LIN {X 0,Y 591.897,Z 1174.931,A -85,B 0,C 180,E1 27089.711,E2 27089.711} C_VEL
LIN {X 0,Y 591.908,Z 1174.109,A -85,B 0,C 180,E1 27087.29,E2 27087.29} C_VEL
LIN {X 0,Y 591.924,Z 1171.503,A -85,B 0,C 180,E1 27084.573,E2 27084.573} C_VEL
LIN {X 0,Y 591.983,Z 1167.392,A -85,B 0,C 180,E1 27082.04,E2 27082.04} C_VEL
LIN {X 0,Y 592.101,Z 1162.202,A -85,B 0,C 180,E1 27079.69,E2 27079.69} C_VEL
LIN {X 0,Y 592.311,Z 1155.916,A -85,B 0,C 180,E1 27077.424,E2 27077.424} C_VEL
LIN {X 0,Y 592.664,Z 1148.61,A -85,B 0,C 180,E1 27075.242,E2 27075.242} C_VEL
LIN {X 0,Y 593.231,Z 1139.207,A -85,B 0,C 180,E1 27072.846,E2 27072.846} C_VEL
LIN {X 0,Y 594.193,Z 1126.707,A -85,B 0,C 180,E1 27070.165,E2 27070.165} C_VEL
LIN {X 0,Y 595.161,Z 1115.669,A -85,B 0,C 180,E1 27068.103,E2 27068.103} C_VEL
LIN {X 0,Y 596.322,Z 1104.081,A -85,B 0,C 180,E1 27066.167,E2 27066.167} C_VEL
LIN {X 0,Y 597.667,Z 1091.843,A -85,B 0,C 180,E1 27064.324,E2 27064.324} C_VEL
LIN {X 0,Y 599.411,Z 1077.454,A -85,B 0,C 180,E1 27062.373,E2 27062.373} C_VEL
LIN {X 0,Y 601.826,Z 1058.389,A -85,B 0,C 180,E1 27060.068,E2 27060.068} C_VEL
LIN {X 0,Y 604.426,Z 1038.878,A -85,B 0,C 180,E1 27058.01,E2 27058.01} C_VEL
LIN {X 0,Y 606.926,Z 1020.464,A -85,B 0,C 180,E1 27056.278,E2 27056.278} C_VEL
LIN {X 0,Y 609.509,Z 1001.423,A -85,B 0,C 180,E1 27054.673,E2 27054.673} C_VEL
LIN {X 0,Y 612.678,Z 977.882,A -85,B 0,C 180,E1 27052.921,E2 27052.921} C_VEL
LIN {X 0,Y 615.57,Z 955.308,A -85,B 0,C 180,E1 27051.472,E2 27051.472} C_VEL
LIN {X 0,Y 618.014,Z 935.338,A -85,B 0,C 180,E1 27050.34,E2 27050.34} C_VEL
LIN {X 0,Y 620.241,Z 915.853,A -85,B 0,C 180,E1 27049.364,E2 27049.364} C_VEL
LIN {X 0,Y 622.411,Z 895.48,A -85,B 0,C 180,E1 27048.471,E2 27048.471} C_VEL
LIN {X 0,Y 624.359,Z 875.247,A -85,B 0,C 180,E1 27047.705,E2 27047.705} C_VEL
LIN {X 0,Y 626.22,Z 853.565,A -85,B 0,C 180,E1 27047.01,E2 27047.01} C_VEL
LIN {X 0,Y 627.748,Z 832.2,A -85,B 0,C 180,E1 27046.449,E2 27046.449} C_VEL
LIN {X 0,Y 629.027,Z 806.934,A -85,B 0,C 180,E1 27045.948,E2 27045.948} C_VEL
LIN {X 0,Y 629.985,Z 765.209,A -85,B 0,C 180,E1 27045.381,E2 27045.381} C_VEL
LIN {X 0,Y 632.547,Z 636.89,A -85,B 0,C 180,E1 27043.662,E2 27043.662} C_VEL
LIN {X 0,Y 637.374,Z 475.557,A -85,B 0,C 180,E1 27041.338,E2 27041.338} C_VEL
LIN {X 0,Y 639.96,Z 392.388,A -85,B 0,C 180,E1 27040.129,E2 27040.129} C_VEL
LIN {X 0,Y 636.531,Z 387.853,A -85,B 0,C 180,E1 27039.678,E2 27039.678} C_VEL
LIN {X 0,Y 622.331,Z 374.151,A -85,B 0,C 180,E1 27037.803,E2 27037.803} C_VEL
LIN {X 0,Y 613.97,Z 366.431,A -85,B 0,C 180,E1 27036.624,E2 27036.624} C_VEL
LIN {X 0,Y 611.495,Z 361.898,A -85,B 0,C 180,E1 27035.323,E2 27035.323} C_VEL
LIN {X 0,Y 608.852,Z 357.084,A -85,B 0,C 180,E1 27033.83,E2 27033.83} C_VEL
LIN {X 0,Y 606.547,Z 352.971,A -85,B 0,C 180,E1 27032.435,E2 27032.435} C_VEL
LIN {X 0,Y 605.226,Z 351.161,A -85,B 0,C 180,E1 27031.693,E2 27031.693} C_VEL
LIN {X 0,Y 602.949,Z 346.733,A -85,B 0,C 180,E1 27030.047,E2 27030.047} C_VEL
LIN {X 0,Y 600.511,Z 343.051,A -85,B 0,C 180,E1 27028.33,E2 27028.33} C_VEL
LIN {X 0,Y 599.929,Z 341.473,A -85,B 0,C 180,E1 27027.711,E2 27027.711} C_VEL
LIN {X 0,Y 597.262,Z 337.966,A -85,B 0,C 180,E1 27025.59,E2 27025.59} C_VEL
LIN {X 0,Y 596.525,Z 335.866,A -85,B 0,C 180,E1 27024.563,E2 27024.563} C_VEL
LIN {X 0,Y 593.473,Z 331.614,A -85,B 0,C 180,E1 27020.927,E2 27020.927} C_VEL
LIN {X 0,Y 593.167,Z 330.296,A -85,B 0,C 180,E1 27019.805,E2 27019.805} C_VEL
LIN {X 0,Y 593.177,Z 330.306,A -85,B 0,C 180,E1 27016.652,E2 27016.652} C_VEL
LIN {X 0,Y 593.194,Z 330.338,A -85,B 0,C 180,E1 27013.451,E2 27013.451} C_VEL
LIN {X 0,Y 593.184,Z 330.295,A -85,B 0,C 180,E1 27010.097,E2 27010.097} C_VEL
LIN {X 0,Y 593.196,Z 330.521,A -85,B 0,C 180,E1 27008.14,E2 27008.14} C_VEL
LIN {X 0,Y 596.195,Z 335.653,A -85,B 0,C 180,E1 27003.943,E2 27003.943} C_VEL
LIN {X 0,Y 596.833,Z 336.421,A -85,B 0,C 180,E1 27003.362,E2 27003.362} C_VEL
LIN {X 0,Y 598.756,Z 340.365,A -85,B 0,C 180,E1 27001.34,E2 27001.34} C_VEL
LIN {X 0,Y 600.215,Z 341.797,A -85,B 0,C 180,E1 27000.382,E2 27000.382} C_VEL
LIN {X 0,Y 601.93,Z 345.619,A -85,B 0,C 180,E1 26998.858,E2 26998.858} C_VEL
LIN {X 0,Y 603.535,Z 347.505,A -85,B 0,C 180,E1 26997.911,E2 26997.911} C_VEL
LIN {X 0,Y 605.549,Z 351.442,A -85,B 0,C 180,E1 26996.497,E2 26996.497} C_VEL
LIN {X 0,Y 606.629,Z 352.745,A -85,B 0,C 180,E1 26995.936,E2 26995.936} C_VEL
LIN {X 0,Y 608.729,Z 356.813,A -85,B 0,C 180,E1 26994.628,E2 26994.628} C_VEL
LIN {X 0,Y 609.804,Z 358.433,A -85,B 0,C 180,E1 26994.071,E2 26994.071} C_VEL
LIN {X 0,Y 612.046,Z 362.396,A -85,B 0,C 180,E1 26992.868,E2 26992.868} C_VEL
LIN {X 0,Y 615.694,Z 369.01,A -85,B 0,C 180,E1 26991.031,E2 26991.031} C_VEL
LIN {X 0,Y 618.78,Z 374.761,A -85,B 0,C 180,E1 26989.573,E2 26989.573} C_VEL
LIN {X 0,Y 621.416,Z 379.7,A -85,B 0,C 180,E1 26988.397,E2 26988.397} C_VEL
LIN {X 0,Y 625.72,Z 387.719,A -85,B 0,C 180,E1 26986.602,E2 26986.602} C_VEL
LIN {X 0,Y 632.277,Z 400.596,A -85,B 0,C 180,E1 26984.028,E2 26984.028} C_VEL
LIN {X 0,Y 638.414,Z 413.491,A -85,B 0,C 180,E1 26981.745,E2 26981.745} C_VEL
LIN {X 0,Y 634.586,Z 446.496,A -85,B 0,C 180,E1 26978.994,E2 26978.994} C_VEL
LIN {X 0,Y 630.632,Z 482.853,A -85,B 0,C 180,E1 26976.102,E2 26976.102} C_VEL
LIN {X 0,Y 626.774,Z 520.74,A -85,B 0,C 180,E1 26973.213,E2 26973.213} C_VEL
LIN {X 0,Y 622.971,Z 560.912,A -85,B 0,C 180,E1 26970.26,E2 26970.26} C_VEL
LIN {X 0,Y 622.003,Z 580.567,A -85,B 0,C 180,E1 26968.779,E2 26968.779} C_VEL
LIN {X 0,Y 622.974,Z 596.183,A -85,B 0,C 180,E1 26967.474,E2 26967.474} C_VEL
LIN {X 0,Y 625.659,Z 609.898,A -85,B 0,C 180,E1 26966.202,E2 26966.202} C_VEL
LIN {X 0,Y 630.378,Z 623.068,A -85,B 0,C 180,E1 26964.845,E2 26964.845} C_VEL
LIN {X 0,Y 637.026,Z 634.807,A -85,B 0,C 180,E1 26963.495,E2 26963.495} C_VEL
LIN {X 0,Y 644.492,Z 643.967,A -85,B 0,C 180,E1 26962.319,E2 26962.319} C_VEL
LIN {X 0,Y 654.158,Z 652.543,A -85,B 0,C 180,E1 26961.081,E2 26961.081} C_VEL
LIN {X 0,Y 665.614,Z 659.76,A -85,B 0,C 180,E1 26959.875,E2 26959.875} C_VEL
LIN {X 0,Y 678.93,Z 665.442,A -85,B 0,C 180,E1 26958.716,E2 26958.716} C_VEL
LIN {X 0,Y 684.652,Z 667.08,A -85,B 0,C 180,E1 26958.244,E2 26958.244} C_VEL
LIN {X 0,Y 688.639,Z 667.261,A -85,B 0,C 180,E1 26957.757,E2 26957.757} C_VEL
LIN {X 0,Y 691.101,Z 666.327,A -85,B 0,C 180,E1 26957.269,E2 26957.269} C_VEL
LIN {X 0,Y 692.176,Z 664.764,A -85,B 0,C 180,E1 26956.842,E2 26956.842} C_VEL
LIN {X 0,Y 684.254,Z 680.558,A -85,B 0,C 180,E1 26956.877,E2 26956.877} C_VEL
LIN {X 0,Y 674.402,Z 696.32,A -85,B 0,C 180,E1 26956.838,E2 26956.838} C_VEL
LIN {X 0,Y 664.605,Z 710.324,A -85,B 0,C 180,E1 26956.682,E2 26956.682} C_VEL
LIN {X 0,Y 657.671,Z 721.169,A -85,B 0,C 180,E1 26956.42,E2 26956.42} C_VEL
LIN {X 0,Y 655.289,Z 724.887,A -85,B 0,C 180,E1 26956.322,E2 26956.322} C_VEL
LIN {X 0,Y 646.984,Z 736.157,A -85,B 0,C 180,E1 26956.067,E2 26956.067} C_VEL
LIN {X 0,Y 640.901,Z 746.673,A -85,B 0,C 180,E1 26955.731,E2 26955.731} C_VEL
LIN {X 0,Y 633.774,Z 760.569,A -85,B 0,C 180,E1 26955.229,E2 26955.229} C_VEL
LIN {X 0,Y 631.455,Z 766.233,A -85,B 0,C 180,E1 26955.02,E2 26955.02} C_VEL
LIN {X 0,Y 629.635,Z 829.003,A -85,B 0,C 180,E1 26954.165,E2 26954.165} C_VEL
LIN {X 0,Y 628.095,Z 857.233,A -85,B 0,C 180,E1 26953.624,E2 26953.624} C_VEL
LIN {X 0,Y 626.337,Z 882.698,A -85,B 0,C 180,E1 26952.976,E2 26952.976} C_VEL
LIN {X 0,Y 624.168,Z 907.973,A -85,B 0,C 180,E1 26952.159,E2 26952.159} C_VEL
LIN {X 0,Y 621.785,Z 932.13,A -85,B 0,C 180,E1 26951.208,E2 26951.208} C_VEL
LIN {X 0,Y 619.008,Z 957.322,A -85,B 0,C 180,E1 26950.034,E2 26950.034} C_VEL
LIN {X 0,Y 616.244,Z 980.499,A -85,B 0,C 180,E1 26948.776,E2 26948.776} C_VEL
LIN {X 0,Y 613.147,Z 1004.437,A -85,B 0,C 180,E1 26947.268,E2 26947.268} C_VEL
LIN {X 0,Y 610.013,Z 1027.671,A -85,B 0,C 180,E1 26945.582,E2 26945.582} C_VEL
LIN {X 0,Y 607.148,Z 1048.872,A -85,B 0,C 180,E1 26943.822,E2 26943.822} C_VEL
LIN {X 0,Y 604.324,Z 1069.852,A -85,B 0,C 180,E1 26941.855,E2 26941.855} C_VEL
LIN {X 0,Y 601.773,Z 1088.672,A -85,B 0,C 180,E1 26939.848,E2 26939.848} C_VEL
LIN {X 0,Y 599.465,Z 1107.176,A -85,B 0,C 180,E1 26937.624,E2 26937.624} C_VEL
LIN {X 0,Y 597.623,Z 1122.284,A -85,B 0,C 180,E1 26935.571,E2 26935.571} C_VEL
LIN {X 0,Y 595.98,Z 1137.726,A -85,B 0,C 180,E1 26933.218,E2 26933.218} C_VEL
LIN {X 0,Y 594.582,Z 1152.188,A -85,B 0,C 180,E1 26930.679,E2 26930.679} C_VEL
LIN {X 0,Y 593.639,Z 1163.642,A -85,B 0,C 180,E1 26928.358,E2 26928.358} C_VEL
LIN {X 0,Y 592.868,Z 1174.752,A -85,B 0,C 180,E1 26925.754,E2 26925.754} C_VEL
LIN {X 0,Y 592.395,Z 1184.279,A -85,B 0,C 180,E1 26923.071,E2 26923.071} C_VEL
LIN {X 0,Y 592.116,Z 1191.662,A -85,B 0,C 180,E1 26920.507,E2 26920.507} C_VEL
LIN {X 0,Y 591.985,Z 1197.33,A -85,B 0,C 180,E1 26917.96,E2 26917.96} C_VEL
LIN {X 0,Y 591.928,Z 1201.413,A -85,B 0,C 180,E1 26915.427,E2 26915.427} C_VEL
LIN {X 0,Y 591.915,Z 1203.98,A -85,B 0,C 180,E1 26912.904,E2 26912.904} C_VEL
LIN {X 0,Y 591.893,Z 1204.916,A -85,B 0,C 180,E1 26910.483,E2 26910.483} C_VEL
LIN {X 0,Y 591.912,Z 1204.414,A -85,B 0,C 180,E1 26907.869,E2 26907.869} C_VEL
LIN {X 0,Y 591.917,Z 1202.356,A -85,B 0,C 180,E1 26905.314,E2 26905.314} C_VEL
LIN {X 0,Y 591.963,Z 1198.771,A -85,B 0,C 180,E1 26902.819,E2 26902.819} C_VEL
LIN {X 0,Y 592.063,Z 1193.554,A -85,B 0,C 180,E1 26900.276,E2 26900.276} C_VEL
LIN {X 0,Y 592.274,Z 1186.734,A -85,B 0,C 180,E1 26897.717,E2 26897.717} C_VEL
LIN {X 0,Y 592.658,Z 1178.841,A -85,B 0,C 180,E1 26895.34,E2 26895.34} C_VEL
LIN {X 0,Y 593.241,Z 1169.012,A -85,B 0,C 180,E1 26892.844,E2 26892.844} C_VEL
LIN {X 0,Y 594.212,Z 1156.49,A -85,B 0,C 180,E1 26890.16,E2 26890.16} C_VEL
LIN {X 0,Y 595.372,Z 1143.738,A -85,B 0,C 180,E1 26887.797,E2 26887.797} C_VEL
LIN {X 0,Y 596.954,Z 1128.582,A -85,B 0,C 180,E1 26885.349,E2 26885.349} C_VEL
LIN {X 0,Y 598.753,Z 1112.617,A -85,B 0,C 180,E1 26883.091,E2 26883.091} C_VEL
LIN {X 0,Y 600.746,Z 1096.868,A -85,B 0,C 180,E1 26881.103,E2 26881.103} C_VEL
LIN {X 0,Y 603.341,Z 1076.831,A -85,B 0,C 180,E1 26878.864,E2 26878.864} C_VEL
LIN {X 0,Y 605.969,Z 1057.522,A -85,B 0,C 180,E1 26876.955,E2 26876.955} C_VEL
LIN {X 0,Y 608.904,Z 1036.067,A -85,B 0,C 180,E1 26875.09,E2 26875.09} C_VEL
LIN {X 0,Y 611.964,Z 1013.202,A -85,B 0,C 180,E1 26873.346,E2 26873.346} C_VEL
LIN {X 0,Y 614.913,Z 990.648,A -85,B 0,C 180,E1 26871.836,E2 26871.836} C_VEL
LIN {X 0,Y 618.022,Z 965.736,A -85,B 0,C 180,E1 26870.398,E2 26870.398} C_VEL
LIN {X 0,Y 620.79,Z 941.484,A -85,B 0,C 180,E1 26869.202,E2 26869.202} C_VEL
LIN {X 0,Y 623.308,Z 916.78,A -85,B 0,C 180,E1 26868.169,E2 26868.169} C_VEL
LIN {X 0,Y 625.72,Z 889.943,A -85,B 0,C 180,E1 26867.242,E2 26867.242} C_VEL
LIN {X 0,Y 627.646,Z 864.672,A -85,B 0,C 180,E1 26866.545,E2 26866.545} C_VEL
LIN {X 0,Y 629.244,Z 837.387,A -85,B 0,C 180,E1 26865.976,E2 26865.976} C_VEL
LIN {X 0,Y 630.409,Z 805.39,A -85,B 0,C 180,E1 26865.494,E2 26865.494} C_VEL
LIN {X 0,Y 631.728,Z 755.195,A -85,B 0,C 180,E1 26864.798,E2 26864.798} C_VEL
LIN {X 0,Y 639.334,Z 659.968,A -85,B 0,C 180,E1 26863.211,E2 26863.211} C_VEL
LIN {X 0,Y 640.721,Z 644.342,A -85,B 0,C 180,E1 26862.962,E2 26862.962} C_VEL
LIN {X 0,Y 643.607,Z 611.399,A -85,B 0,C 180,E1 26862.434,E2 26862.434} C_VEL
LIN {X 0,Y 645.463,Z 593.682,A -85,B 0,C 180,E1 26862.178,E2 26862.178} C_VEL
LIN {X 0,Y 647.573,Z 567.044,A -85,B 0,C 180,E1 26861.731,E2 26861.731} C_VEL
LIN {X 0,Y 651.175,Z 535.673,A -85,B 0,C 180,E1 26861.308,E2 26861.308} C_VEL
LIN {X 0,Y 652.805,Z 513.097,A -85,B 0,C 180,E1 26860.913,E2 26860.913} C_VEL
LIN {X 0,Y 656.784,Z 480.454,A -85,B 0,C 180,E1 26860.496,E2 26860.496} C_VEL
LIN {X 0,Y 657.711,Z 472.636,A -85,B 0,C 180,E1 26860.394,E2 26860.394} C_VEL
LIN {X 0,Y 658.916,Z 453.469,A -85,B 0,C 180,E1 26860.042,E2 26860.042} C_VEL
LIN {X 0,Y 662.468,Z 423.806,A -85,B 0,C 180,E1 26859.659,E2 26859.659} C_VEL
LIN {X 0,Y 662.806,Z 420.787,A -85,B 0,C 180,E1 26859.618,E2 26859.618} C_VEL
LIN {X 0,Y 654.528,Z 413.473,A -85,B 0,C 180,E1 26858.612,E2 26858.612} C_VEL
LIN {X 0,Y 646.489,Z 404.608,A -85,B 0,C 180,E1 26857.545,E2 26857.545} C_VEL
LIN {X 0,Y 630.725,Z 381.497,A -85,B 0,C 180,E1 26855.132,E2 26855.132} C_VEL
LIN {X 0,Y 618.485,Z 364.345,A -85,B 0,C 180,E1 26853.095,E2 26853.095} C_VEL
LIN {X 0,Y 609.724,Z 352.82,A -85,B 0,C 180,E1 26851.543,E2 26851.543} C_VEL
LIN {X 0,Y 605.772,Z 347.565,A -85,B 0,C 180,E1 26850.804,E2 26850.804} C_VEL
LIN {X 0,Y 602.767,Z 343.666,A -85,B 0,C 180,E1 26850.229,E2 26850.229} C_VEL
LIN {X 0,Y 601.685,Z 342.131,A -85,B 0,C 180,E1 26850.014,E2 26850.014} C_VEL
LIN {X 0,Y 598.782,Z 338.928,A -85,B 0,C 180,E1 26849.458,E2 26849.458} C_VEL
LIN {X 0,Y 597.371,Z 336.419,A -85,B 0,C 180,E1 26849.149,E2 26849.149} C_VEL
LIN {X 0,Y 594.578,Z 333.934,A -85,B 0,C 180,E1 26848.614,E2 26848.614} C_VEL
LIN {X 0,Y 593.298,Z 330.916,A -85,B 0,C 180,E1 26848.296,E2 26848.296} C_VEL
LIN {X 0,Y 593.203,Z 330.343,A -85,B 0,C 180,E1 26848.241,E2 26848.241} C_VEL
LIN {X 0,Y 593.175,Z 330.268,A -85,B 0,C 180,E1 26844.921,E2 26844.921} C_VEL
LIN {X 0,Y 593.175,Z 330.342,A -85,B 0,C 180,E1 26841.751,E2 26841.751} C_VEL
LIN {X 0,Y 593.178,Z 330.344,A -85,B 0,C 180,E1 26838.578,E2 26838.578} C_VEL
LIN {X 0,Y 593.172,Z 330.346,A -85,B 0,C 180,E1 26835.376,E2 26835.376} C_VEL
LIN {X 0,Y 593.222,Z 330.489,A -85,B 0,C 180,E1 26834.159,E2 26834.159} C_VEL
LIN {X 0,Y 597.978,Z 346.498,A -85,B 0,C 180,E1 26833.44,E2 26833.44} C_VEL
LIN {X 0,Y 597.928,Z 424.43,A -85,B 0,C 180,E1 26830.722,E2 26830.722} C_VEL
LIN {X 0,Y 598.267,Z 504.666,A -85,B 0,C 180,E1 26827.78,E2 26827.78} C_VEL
LIN {X 0,Y 598.24,Z 578.346,A -85,B 0,C 180,E1 26824.986,E2 26824.986} C_VEL
LIN {X 0,Y 597.772,Z 656.038,A -85,B 0,C 180,E1 26821.965,E2 26821.965} C_VEL
LIN {X 0,Y 597.006,Z 735.74,A -85,B 0,C 180,E1 26818.8,E2 26818.8} C_VEL
LIN {X 0,Y 596.103,Z 814.288,A -85,B 0,C 180,E1 26815.623,E2 26815.623} C_VEL
LIN {X 0,Y 595.528,Z 847.719,A -85,B 0,C 180,E1 26814.267,E2 26814.267} C_VEL
LIN {X 0,Y 595.129,Z 853.977,A -85,B 0,C 180,E1 26814.046,E2 26814.046} C_VEL
LIN {X 0,Y 594.541,Z 967.975,A -85,B 0,C 180,E1 26812.596,E2 26812.596} C_VEL
LIN {X 0,Y 594.552,Z 980.318,A -85,B 0,C 180,E1 26812.313,E2 26812.313} C_VEL
LIN {X 0,Y 594.512,Z 991.961,A -85,B 0,C 180,E1 26811.927,E2 26811.927} C_VEL
LIN {X 0,Y 594.401,Z 1005.064,A -85,B 0,C 180,E1 26811.341,E2 26811.341} C_VEL
LIN {X 0,Y 594.177,Z 1017.894,A -85,B 0,C 180,E1 26810.556,E2 26810.556} C_VEL
LIN {X 0,Y 593.986,Z 1027.459,A -85,B 0,C 180,E1 26809.819,E2 26809.819} C_VEL
LIN {X 0,Y 593.777,Z 1035.869,A -85,B 0,C 180,E1 26809.03,E2 26809.03} C_VEL
LIN {X 0,Y 593.569,Z 1043.67,A -85,B 0,C 180,E1 26808.14,E2 26808.14} C_VEL
LIN {X 0,Y 593.36,Z 1051.4,A -85,B 0,C 180,E1 26807.049,E2 26807.049} C_VEL
LIN {X 0,Y 593.145,Z 1058.271,A -85,B 0,C 180,E1 26805.752,E2 26805.752} C_VEL
LIN {X 0,Y 593.025,Z 1062.584,A -85,B 0,C 180,E1 26804.65,E2 26804.65} C_VEL
LIN {X 0,Y 592.933,Z 1065.672,A -85,B 0,C 180,E1 26803.542,E2 26803.542} C_VEL
LIN {X 0,Y 592.879,Z 1067.603,A -85,B 0,C 180,E1 26802.429,E2 26802.429} C_VEL
LIN {X 0,Y 592.841,Z 1068.45,A -85,B 0,C 180,E1 26801.207,E2 26801.207} C_VEL
LIN {X 0,Y 592.845,Z 1067.619,A -85,B 0,C 180,E1 26799.669,E2 26799.669} C_VEL
LIN {X 0,Y 592.869,Z 1065.357,A -85,B 0,C 180,E1 26798.428,E2 26798.428} C_VEL
LIN {X 0,Y 592.936,Z 1062.021,A -85,B 0,C 180,E1 26797.283,E2 26797.283} C_VEL
LIN {X 0,Y 593.038,Z 1057.325,A -85,B 0,C 180,E1 26796.131,E2 26796.131} C_VEL
LIN {X 0,Y 593.245,Z 1049.74,A -85,B 0,C 180,E1 26794.759,E2 26794.759} C_VEL
LIN {X 0,Y 593.451,Z 1041.883,A -85,B 0,C 180,E1 26793.684,E2 26793.684} C_VEL
LIN {X 0,Y 593.673,Z 1033.295,A -85,B 0,C 180,E1 26792.734,E2 26792.734} C_VEL
LIN {X 0,Y 593.952,Z 1022.469,A -85,B 0,C 180,E1 26791.767,E2 26791.767} C_VEL
LIN {X 0,Y 594.193,Z 1009.805,A -85,B 0,C 180,E1 26790.901,E2 26790.901} C_VEL
LIN {X 0,Y 594.373,Z 998.89,A -85,B 0,C 180,E1 26790.313,E2 26790.313} C_VEL
LIN {X 0,Y 594.504,Z 987.303,A -85,B 0,C 180,E1 26789.825,E2 26789.825} C_VEL
LIN {X 0,Y 594.602,Z 972.83,A -85,B 0,C 180,E1 26789.383,E2 26789.383} C_VEL
LIN {X 0,Y 594.58,Z 956.069,A -85,B 0,C 180,E1 26789.096,E2 26789.096} C_VEL
LIN {X 0,Y 595.087,Z 870.743,A -85,B 0,C 180,E1 26788.038,E2 26788.038} C_VEL
LIN {X 0,Y 594.247,Z 865.604,A -85,B 0,C 180,E1 26787.949,E2 26787.949} C_VEL
LIN {X 0,Y 587.888,Z 851.327,A -85,B 0,C 180,E1 26787.624,E2 26787.624} C_VEL
LIN {X 0,Y 587.567,Z 848.543,A -85,B 0,C 180,E1 26787.539,E2 26787.539} C_VEL
LIN {X 0,Y 588.582,Z 796.208,A -85,B 0,C 180,E1 26785.342,E2 26785.342} C_VEL
LIN {X 0,Y 589.928,Z 714.708,A -85,B 0,C 180,E1 26781.905,E2 26781.905} C_VEL
LIN {X 0,Y 590.88,Z 660.354,A -85,B 0,C 180,E1 26779.6,E2 26779.6} C_VEL
LIN {X 0,Y 592.005,Z 661.931,A -85,B 0,C 180,E1 26779.438,E2 26779.438} C_VEL
LIN {X 0,Y 593.686,Z 661.837,A -85,B 0,C 180,E1 26779.26,E2 26779.26} C_VEL
LIN {X 0,Y 596.517,Z 659.34,A -85,B 0,C 180,E1 26779.018,E2 26779.018} C_VEL
LIN {X 0,Y 600.352,Z 653.293,A -85,B 0,C 180,E1 26778.759,E2 26778.759} C_VEL
LIN {X 0,Y 604.334,Z 651.507,A -85,B 0,C 180,E1 26778.4,E2 26778.4} C_VEL
LIN {X 0,Y 608.324,Z 647.655,A -85,B 0,C 180,E1 26778.106,E2 26778.106} C_VEL
LIN {X 0,Y 611.151,Z 643.737,A -85,B 0,C 180,E1 26777.935,E2 26777.935} C_VEL
LIN {X 0,Y 615.844,Z 641.07,A -85,B 0,C 180,E1 26777.576,E2 26777.576} C_VEL
LIN {X 0,Y 620.545,Z 636.286,A -85,B 0,C 180,E1 26777.253,E2 26777.253} C_VEL
LIN {X 0,Y 622.028,Z 634.442,A -85,B 0,C 180,E1 26777.159,E2 26777.159} C_VEL
LIN {X 0,Y 626.738,Z 631.619,A -85,B 0,C 180,E1 26776.813,E2 26776.813} C_VEL
LIN {X 0,Y 623.646,Z 757.358,A -85,B 0,C 180,E1 26775.063,E2 26775.063} C_VEL
LIN {X 0,Y 622.408,Z 807.519,A -85,B 0,C 180,E1 26774.37,E2 26774.37} C_VEL
LIN {X 0,Y 621.009,Z 834.635,A -85,B 0,C 180,E1 26773.828,E2 26773.828} C_VEL
LIN {X 0,Y 619.62,Z 856.522,A -85,B 0,C 180,E1 26773.27,E2 26773.27} C_VEL
LIN {X 0,Y 618.179,Z 876.153,A -85,B 0,C 180,E1 26772.667,E2 26772.667} C_VEL
LIN {X 0,Y 616.582,Z 893.157,A -85,B 0,C 180,E1 26772.036,E2 26772.036} C_VEL
LIN {X 0,Y 614.249,Z 914.189,A -85,B 0,C 180,E1 26771.121,E2 26771.121} C_VEL
LIN {X 0,Y 612.021,Z 932.876,A -85,B 0,C 180,E1 26770.191,E2 26770.191} C_VEL
LIN {X 0,Y 609.654,Z 951.359,A -85,B 0,C 180,E1 26769.157,E2 26769.157} C_VEL
LIN {X 0,Y 607.2,Z 969.562,A -85,B 0,C 180,E1 26768.016,E2 26768.016} C_VEL
LIN {X 0,Y 604.707,Z 987.416,A -85,B 0,C 180,E1 26766.768,E2 26766.768} C_VEL
LIN {X 0,Y 602.162,Z 1005.245,A -85,B 0,C 180,E1 26765.382,E2 26765.382} C_VEL
LIN {X 0,Y 599.527,Z 1023.571,A -85,B 0,C 180,E1 26763.795,E2 26763.795} C_VEL
LIN {X 0,Y 596.613,Z 1043.916,A -85,B 0,C 180,E1 26761.82,E2 26761.82} C_VEL
LIN {X 0,Y 593.869,Z 1063.27,A -85,B 0,C 180,E1 26759.671,E2 26759.671} C_VEL
LIN {X 0,Y 591.859,Z 1078.36,A -85,B 0,C 180,E1 26757.794,E2 26757.794} C_VEL
LIN {X 0,Y 590.022,Z 1092.656,A -85,B 0,C 180,E1 26755.82,E2 26755.82} C_VEL
LIN {X 0,Y 588.463,Z 1106.104,A -85,B 0,C 180,E1 26753.748,E2 26753.748} C_VEL
LIN {X 0,Y 586.878,Z 1121.364,A -85,B 0,C 180,E1 26751.07,E2 26751.07} C_VEL
LIN {X 0,Y 585.862,Z 1132.457,A -85,B 0,C 180,E1 26748.819,E2 26748.819} C_VEL
LIN {X 0,Y 585.18,Z 1141.293,A -85,B 0,C 180,E1 26746.785,E2 26746.785} C_VEL
LIN {X 0,Y 584.683,Z 1149.344,A -85,B 0,C 180,E1 26744.662,E2 26744.662} C_VEL
LIN {X 0,Y 584.329,Z 1156.234,A -85,B 0,C 180,E1 26742.553,E2 26742.553} C_VEL
LIN {X 0,Y 584.112,Z 1162.464,A -85,B 0,C 180,E1 26740.256,E2 26740.256} C_VEL
LIN {X 0,Y 583.989,Z 1167.597,A -85,B 0,C 180,E1 26737.874,E2 26737.874} C_VEL
LIN {X 0,Y 583.927,Z 1171.885,A -85,B 0,C 180,E1 26735.11,E2 26735.11} C_VEL
LIN {X 0,Y 583.907,Z 1174.164,A -85,B 0,C 180,E1 26732.553,E2 26732.553} C_VEL
LIN {X 0,Y 583.901,Z 1174.928,A -85,B 0,C 180,E1 26730.197,E2 26730.197} C_VEL
LIN {X 0,Y 583.911,Z 1174.355,A -85,B 0,C 180,E1 26727.744,E2 26727.744} C_VEL
LIN {X 0,Y 583.915,Z 1172.492,A -85,B 0,C 180,E1 26725.385,E2 26725.385} C_VEL
LIN {X 0,Y 583.954,Z 1169.172,A -85,B 0,C 180,E1 26722.92,E2 26722.92} C_VEL
LIN {X 0,Y 584.072,Z 1163.675,A -85,B 0,C 180,E1 26720.144,E2 26720.144} C_VEL
LIN {X 0,Y 584.291,Z 1157.111,A -85,B 0,C 180,E1 26717.65,E2 26717.65} C_VEL
LIN {X 0,Y 584.636,Z 1150.02,A -85,B 0,C 180,E1 26715.44,E2 26715.44} C_VEL
LIN {X 0,Y 585.13,Z 1142.068,A -85,B 0,C 180,E1 26713.318,E2 26713.318} C_VEL
LIN {X 0,Y 585.792,Z 1133.335,A -85,B 0,C 180,E1 26711.284,E2 26711.284} C_VEL
LIN {X 0,Y 586.614,Z 1123.912,A -85,B 0,C 180,E1 26709.341,E2 26709.341} C_VEL
LIN {X 0,Y 587.671,Z 1113.33,A -85,B 0,C 180,E1 26707.387,E2 26707.387} C_VEL
LIN {X 0,Y 589.142,Z 1100.183,A -85,B 0,C 180,E1 26705.217,E2 26705.217} C_VEL
LIN {X 0,Y 591.339,Z 1082.2,A -85,B 0,C 180,E1 26702.62,E2 26702.62} C_VEL
LIN {X 0,Y 593.428,Z 1066.615,A -85,B 0,C 180,E1 26700.64,E2 26700.64} C_VEL
LIN {X 0,Y 595.625,Z 1050.692,A -85,B 0,C 180,E1 26698.819,E2 26698.819} C_VEL
LIN {X 0,Y 598.392,Z 1031.392,A -85,B 0,C 180,E1 26696.841,E2 26696.841} C_VEL
LIN {X 0,Y 601.593,Z 1009.292,A -85,B 0,C 180,E1 26694.86,E2 26694.86} C_VEL
LIN {X 0,Y 604.36,Z 989.93,A -85,B 0,C 180,E1 26693.328,E2 26693.328} C_VEL
LIN {X 0,Y 606.925,Z 971.551,A -85,B 0,C 180,E1 26692.026,E2 26692.026} C_VEL
LIN {X 0,Y 609.36,Z 953.557,A -85,B 0,C 180,E1 26690.884,E2 26690.884} C_VEL
LIN {X 0,Y 611.705,Z 935.317,A -85,B 0,C 180,E1 26689.848,E2 26689.848} C_VEL
LIN {X 0,Y 614.049,Z 915.832,A -85,B 0,C 180,E1 26688.866,E2 26688.866} C_VEL
LIN {X 0,Y 616.241,Z 896.216,A -85,B 0,C 180,E1 26687.999,E2 26687.999} C_VEL
LIN {X 0,Y 617.87,Z 879.929,A -85,B 0,C 180,E1 26687.373,E2 26687.373} C_VEL
LIN {X 0,Y 619.415,Z 859.522,A -85,B 0,C 180,E1 26686.725,E2 26686.725} C_VEL
LIN {X 0,Y 620.797,Z 838.049,A -85,B 0,C 180,E1 26686.164,E2 26686.164} C_VEL
LIN {X 0,Y 621.872,Z 817.652,A -85,B 0,C 180,E1 26685.73,E2 26685.73} C_VEL
LIN {X 0,Y 622.665,Z 798.147,A -85,B 0,C 180,E1 26685.403,E2 26685.403} C_VEL
LIN {X 0,Y 626.399,Z 642.254,A -85,B 0,C 180,E1 26683.253,E2 26683.253} C_VEL
LIN {X 0,Y 634.16,Z 414.07,A -85,B 0,C 180,E1 26679.889,E2 26679.889} C_VEL
LIN {X 0,Y 634.628,Z 396.39,A -85,B 0,C 180,E1 26679.621,E2 26679.621} C_VEL
LIN {X 0,Y 632.055,Z 393.601,A -85,B 0,C 180,E1 26679.286,E2 26679.286} C_VEL
LIN {X 0,Y 619.781,Z 381.516,A -85,B 0,C 180,E1 26677.636,E2 26677.636} C_VEL
LIN {X 0,Y 611.282,Z 373.672,A -85,B 0,C 180,E1 26676.425,E2 26676.425} C_VEL
LIN {X 0,Y 608.132,Z 370.809,A -85,B 0,C 180,E1 26675.943,E2 26675.943} C_VEL
LIN {X 0,Y 606.822,Z 368.308,A -85,B 0,C 180,E1 26675.22,E2 26675.22} C_VEL
LIN {X 0,Y 604.105,Z 363.41,A -85,B 0,C 180,E1 26673.675,E2 26673.675} C_VEL
LIN {X 0,Y 601.839,Z 359.085,A -85,B 0,C 180,E1 26672.229,E2 26672.229} C_VEL
LIN {X 0,Y 599.198,Z 354.948,A -85,B 0,C 180,E1 26670.568,E2 26670.568} C_VEL
LIN {X 0,Y 598.463,Z 353.328,A -85,B 0,C 180,E1 26669.971,E2 26669.971} C_VEL
LIN {X 0,Y 596.055,Z 349.621,A -85,B 0,C 180,E1 26668.233,E2 26668.233} C_VEL
LIN {X 0,Y 595.332,Z 347.979,A -85,B 0,C 180,E1 26667.53,E2 26667.53} C_VEL
LIN {X 0,Y 592.79,Z 344.325,A -85,B 0,C 180,E1 26665.368,E2 26665.368} C_VEL
LIN {X 0,Y 592.163,Z 342.565,A -85,B 0,C 180,E1 26664.483,E2 26664.483} C_VEL
LIN {X 0,Y 589.172,Z 338.216,A -85,B 0,C 180,E1 26660.76,E2 26660.76} C_VEL
LIN {X 0,Y 588.742,Z 336.959,A -85,B 0,C 180,E1 26659.65,E2 26659.65} C_VEL
LIN {X 0,Y 587.04,Z 335.405,A -85,B 0,C 180,E1 26655.005,E2 26655.005} C_VEL
LIN {X 0,Y 587.489,Z 335.904,A -85,B 0,C 180,E1 26651.088,E2 26651.088} C_VEL
LIN {X 0,Y 588.982,Z 337.422,A -85,B 0,C 180,E1 26648.1,E2 26648.1} C_VEL
LIN {X 0,Y 592.051,Z 342.514,A -85,B 0,C 180,E1 26643.874,E2 26643.874} C_VEL
LIN {X 0,Y 592.582,Z 343.466,A -85,B 0,C 180,E1 26643.289,E2 26643.289} C_VEL
LIN {X 0,Y 594.754,Z 347.428,A -85,B 0,C 180,E1 26641.156,E2 26641.156} C_VEL
LIN {X 0,Y 595.851,Z 348.705,A -85,B 0,C 180,E1 26640.385,E2 26640.385} C_VEL
LIN {X 0,Y 597.8,Z 352.589,A -85,B 0,C 180,E1 26638.754,E2 26638.754} C_VEL
LIN {X 0,Y 599.06,Z 354.138,A -85,B 0,C 180,E1 26637.991,E2 26637.991} C_VEL
LIN {X 0,Y 601.26,Z 358.247,A -85,B 0,C 180,E1 26636.472,E2 26636.472} C_VEL
LIN {X 0,Y 602.214,Z 359.757,A -85,B 0,C 180,E1 26635.906,E2 26635.906} C_VEL
LIN {X 0,Y 604.639,Z 363.873,A -85,B 0,C 180,E1 26634.496,E2 26634.496} C_VEL
LIN {X 0,Y 607.579,Z 369.036,A -85,B 0,C 180,E1 26632.894,E2 26632.894} C_VEL
LIN {X 0,Y 611.111,Z 375.716,A -85,B 0,C 180,E1 26631.058,E2 26631.058} C_VEL
LIN {X 0,Y 614.004,Z 381.082,A -85,B 0,C 180,E1 26629.681,E2 26629.681} C_VEL
LIN {X 0,Y 618.347,Z 389.075,A -85,B 0,C 180,E1 26627.77,E2 26627.77} C_VEL
LIN {X 0,Y 625.086,Z 402.367,A -85,B 0,C 180,E1 26624.981,E2 26624.981} C_VEL
LIN {X 0,Y 631.564,Z 415.802,A -85,B 0,C 180,E1 26622.494,E2 26622.494} C_VEL
LIN {X 0,Y 632.751,Z 418.495,A -85,B 0,C 180,E1 26622.038,E2 26622.038} C_VEL
LIN {X 0,Y 628.808,Z 450.791,A -85,B 0,C 180,E1 26619.328,E2 26619.328} C_VEL
LIN {X 0,Y 624.705,Z 486.494,A -85,B 0,C 180,E1 26616.468,E2 26616.468} C_VEL
LIN {X 0,Y 620.615,Z 524.504,A -85,B 0,C 180,E1 26613.546,E2 26613.546} C_VEL
LIN {X 0,Y 616.585,Z 564.906,A -85,B 0,C 180,E1 26610.551,E2 26610.551} C_VEL
LIN {X 0,Y 615.611,Z 583.676,A -85,B 0,C 180,E1 26609.119,E2 26609.119} C_VEL
LIN {X 0,Y 616.536,Z 599.846,A -85,B 0,C 180,E1 26607.753,E2 26607.753} C_VEL
LIN {X 0,Y 619.371,Z 614.497,A -85,B 0,C 180,E1 26606.377,E2 26606.377} C_VEL
LIN {X 0,Y 624.083,Z 627.709,A -85,B 0,C 180,E1 26605,E2 26605} C_VEL
LIN {X 0,Y 630.665,Z 639.502,A -85,B 0,C 180,E1 26603.632,E2 26603.632} C_VEL
LIN {X 0,Y 638.042,Z 648.781,A -85,B 0,C 180,E1 26602.438,E2 26602.438} C_VEL
LIN {X 0,Y 647.588,Z 657.546,A -85,B 0,C 180,E1 26601.18,E2 26601.18} C_VEL
LIN {X 0,Y 658.908,Z 664.997,A -85,B 0,C 180,E1 26599.953,E2 26599.953} C_VEL
LIN {X 0,Y 671.336,Z 670.726,A -85,B 0,C 180,E1 26598.828,E2 26598.828} C_VEL
LIN {X 0,Y 680.797,Z 673.766,A -85,B 0,C 180,E1 26598.067,E2 26598.067} C_VEL
LIN {X 0,Y 684.978,Z 674.105,A -85,B 0,C 180,E1 26597.592,E2 26597.592} C_VEL
LIN {X 0,Y 685.455,Z 674.112,A -85,B 0,C 180,E1 26597.515,E2 26597.515} C_VEL
LIN {X 0,Y 674.505,Z 689.052,A -85,B 0,C 180,E1 26597.453,E2 26597.453} C_VEL
LIN {X 0,Y 661.923,Z 704.601,A -85,B 0,C 180,E1 26597.232,E2 26597.232} C_VEL
LIN {X 0,Y 653.836,Z 716.002,A -85,B 0,C 180,E1 26596.967,E2 26596.967} C_VEL
LIN {X 0,Y 649.863,Z 722.315,A -85,B 0,C 180,E1 26596.789,E2 26596.789} C_VEL
LIN {X 0,Y 641.335,Z 733.878,A -85,B 0,C 180,E1 26596.529,E2 26596.529} C_VEL
LIN {X 0,Y 635.156,Z 744.353,A -85,B 0,C 180,E1 26596.2,E2 26596.2} C_VEL
LIN {X 0,Y 627.217,Z 759.808,A -85,B 0,C 180,E1 26595.639,E2 26595.639} C_VEL
LIN {X 0,Y 626.243,Z 762.541,A -85,B 0,C 180,E1 26595.555,E2 26595.555} C_VEL
LIN {X 0,Y 625.47,Z 772.425,A -85,B 0,C 180,E1 26595.471,E2 26595.471} C_VEL
LIN {X 0,Y 623.944,Z 827.243,A -85,B 0,C 180,E1 26594.703,E2 26594.703} C_VEL
LIN {X 0,Y 622.273,Z 855.617,A -85,B 0,C 180,E1 26594.161,E2 26594.161} C_VEL
LIN {X 0,Y 620.284,Z 882.798,A -85,B 0,C 180,E1 26593.467,E2 26593.467} C_VEL
LIN {X 0,Y 618.078,Z 908.548,A -85,B 0,C 180,E1 26592.641,E2 26592.641} C_VEL
LIN {X 0,Y 615.728,Z 931.388,A -85,B 0,C 180,E1 26591.742,E2 26591.742} C_VEL
LIN {X 0,Y 612.797,Z 956.795,A -85,B 0,C 180,E1 26590.556,E2 26590.556} C_VEL
LIN {X 0,Y 609.827,Z 980.503,A -85,B 0,C 180,E1 26589.262,E2 26589.262} C_VEL
LIN {X 0,Y 606.706,Z 1003.411,A -85,B 0,C 180,E1 26587.81,E2 26587.81} C_VEL
LIN {X 0,Y 603.443,Z 1026.315,A -85,B 0,C 180,E1 26586.147,E2 26586.147} C_VEL
LIN {X 0,Y 600.359,Z 1047.699,A -85,B 0,C 180,E1 26584.372,E2 26584.372} C_VEL
LIN {X 0,Y 597.368,Z 1068.839,A -85,B 0,C 180,E1 26582.384,E2 26582.384} C_VEL
LIN {X 0,Y 594.562,Z 1088.261,A -85,B 0,C 180,E1 26580.297,E2 26580.297} C_VEL
LIN {X 0,Y 592.13,Z 1106.396,A -85,B 0,C 180,E1 26578.106,E2 26578.106} C_VEL
LIN {X 0,Y 590.073,Z 1122.283,A -85,B 0,C 180,E1 26575.923,E2 26575.923} C_VEL
LIN {X 0,Y 588.307,Z 1137.724,A -85,B 0,C 180,E1 26573.539,E2 26573.539} C_VEL
LIN {X 0,Y 586.809,Z 1152.191,A -85,B 0,C 180,E1 26570.965,E2 26570.965} C_VEL
LIN {X 0,Y 585.747,Z 1164.11,A -85,B 0,C 180,E1 26568.511,E2 26568.511} C_VEL
LIN {X 0,Y 584.957,Z 1174.75,A -85,B 0,C 180,E1 26565.973,E2 26565.973} C_VEL
LIN {X 0,Y 584.44,Z 1184.277,A -85,B 0,C 180,E1 26563.252,E2 26563.252} C_VEL
LIN {X 0,Y 584.131,Z 1191.663,A -85,B 0,C 180,E1 26560.652,E2 26560.652} C_VEL
LIN {X 0,Y 583.989,Z 1197.329,A -85,B 0,C 180,E1 26558.07,E2 26558.07} C_VEL
LIN {X 0,Y 583.929,Z 1201.412,A -85,B 0,C 180,E1 26555.501,E2 26555.501} C_VEL
LIN {X 0,Y 583.916,Z 1203.979,A -85,B 0,C 180,E1 26552.943,E2 26552.943} C_VEL
LIN {X 0,Y 583.893,Z 1204.916,A -85,B 0,C 180,E1 26550.489,E2 26550.489} C_VEL
LIN {X 0,Y 583.911,Z 1204.413,A -85,B 0,C 180,E1 26547.84,E2 26547.84} C_VEL
LIN {X 0,Y 583.918,Z 1202.391,A -85,B 0,C 180,E1 26545.282,E2 26545.282} C_VEL
LIN {X 0,Y 583.97,Z 1198.769,A -85,B 0,C 180,E1 26542.72,E2 26542.72} C_VEL
LIN {X 0,Y 584.075,Z 1193.552,A -85,B 0,C 180,E1 26540.142,E2 26540.142} C_VEL
LIN {X 0,Y 584.31,Z 1186.733,A -85,B 0,C 180,E1 26537.547,E2 26537.547} C_VEL
LIN {X 0,Y 584.744,Z 1178.486,A -85,B 0,C 180,E1 26535.035,E2 26535.035} C_VEL
LIN {X 0,Y 585.394,Z 1168.583,A -85,B 0,C 180,E1 26532.504,E2 26532.504} C_VEL
LIN {X 0,Y 586.407,Z 1156.328,A -85,B 0,C 180,E1 26529.852,E2 26529.852} C_VEL
LIN {X 0,Y 587.714,Z 1143.159,A -85,B 0,C 180,E1 26527.386,E2 26527.386} C_VEL
LIN {X 0,Y 589.512,Z 1127.255,A -85,B 0,C 180,E1 26524.802,E2 26524.802} C_VEL
LIN {X 0,Y 591.49,Z 1111.057,A -85,B 0,C 180,E1 26522.516,E2 26522.516} C_VEL
LIN {X 0,Y 593.856,Z 1093.671,A -85,B 0,C 180,E1 26520.32,E2 26520.32} C_VEL
LIN {X 0,Y 596.511,Z 1074.442,A -85,B 0,C 180,E1 26518.196,E2 26518.196} C_VEL
LIN {X 0,Y 599.557,Z 1053.51,A -85,B 0,C 180,E1 26516.149,E2 26516.149} C_VEL
LIN {X 0,Y 602.708,Z 1031.646,A -85,B 0,C 180,E1 26514.269,E2 26514.269} C_VEL
LIN {X 0,Y 605.837,Z 1009.375,A -85,B 0,C 180,E1 26512.601,E2 26512.601} C_VEL
LIN {X 0,Y 608.985,Z 986.501,A -85,B 0,C 180,E1 26511.102,E2 26511.102} C_VEL
LIN {X 0,Y 612.195,Z 961.744,A -85,B 0,C 180,E1 26509.7,E2 26509.7} C_VEL
LIN {X 0,Y 615.047,Z 937.979,A -85,B 0,C 180,E1 26508.543,E2 26508.543} C_VEL
LIN {X 0,Y 617.507,Z 914.255,A -85,B 0,C 180,E1 26507.569,E2 26507.569} C_VEL
LIN {X 0,Y 619.905,Z 887.591,A -85,B 0,C 180,E1 26506.673,E2 26506.673} C_VEL
LIN {X 0,Y 621.996,Z 860.208,A -85,B 0,C 180,E1 26505.942,E2 26505.942} C_VEL
LIN {X 0,Y 623.686,Z 832.533,A -85,B 0,C 180,E1 26505.383,E2 26505.383} C_VEL
LIN {X 0,Y 624.899,Z 797.21,A -85,B 0,C 180,E1 26504.866,E2 26504.866} C_VEL
LIN {X 0,Y 626.19,Z 751.211,A -85,B 0,C 180,E1 26504.227,E2 26504.227} C_VEL
LIN {X 0,Y 633.652,Z 660.134,A -85,B 0,C 180,E1 26502.704,E2 26502.704} C_VEL
LIN {X 0,Y 635.032,Z 644.759,A -85,B 0,C 180,E1 26502.457,E2 26502.457} C_VEL
LIN {X 0,Y 638.008,Z 611.522,A -85,B 0,C 180,E1 26501.923,E2 26501.923} C_VEL
LIN {X 0,Y 639.842,Z 594.136,A -85,B 0,C 180,E1 26501.67,E2 26501.67} C_VEL
LIN {X 0,Y 642.055,Z 567.049,A -85,B 0,C 180,E1 26501.215,E2 26501.215} C_VEL
LIN {X 0,Y 645.629,Z 536.228,A -85,B 0,C 180,E1 26500.798,E2 26500.798} C_VEL
LIN {X 0,Y 647.373,Z 513.052,A -85,B 0,C 180,E1 26500.394,E2 26500.394} C_VEL
LIN {X 0,Y 651.452,Z 480.082,A -85,B 0,C 180,E1 26499.974,E2 26499.974} C_VEL
LIN {X 0,Y 652.249,Z 473.101,A -85,B 0,C 180,E1 26499.879,E2 26499.879} C_VEL
LIN {X 0,Y 653.585,Z 453.267,A -85,B 0,C 180,E1 26499.517,E2 26499.517} C_VEL
LIN {X 0,Y 656.819,Z 425.778,A -85,B 0,C 180,E1 26499.153,E2 26499.153} C_VEL
LIN {X 0,Y 645.344,Z 414.407,A -85,B 0,C 180,E1 26497.679,E2 26497.679} C_VEL
LIN {X 0,Y 638.653,Z 405.195,A -85,B 0,C 180,E1 26496.704,E2 26496.704} C_VEL
LIN {X 0,Y 625.051,Z 385.145,A -85,B 0,C 180,E1 26494.548,E2 26494.548} C_VEL
LIN {X 0,Y 614.266,Z 370.144,A -85,B 0,C 180,E1 26492.713,E2 26492.713} C_VEL
LIN {X 0,Y 606.187,Z 359.352,A -85,B 0,C 180,E1 26491.249,E2 26491.249} C_VEL
LIN {X 0,Y 602.382,Z 354.271,A -85,B 0,C 180,E1 26490.526,E2 26490.526} C_VEL
LIN {X 0,Y 599.108,Z 349.769,A -85,B 0,C 180,E1 26489.88,E2 26489.88} C_VEL
LIN {X 0,Y 595.371,Z 345.396,A -85,B 0,C 180,E1 26489.146,E2 26489.146} C_VEL
LIN {X 0,Y 594.142,Z 343.451,A -85,B 0,C 180,E1 26488.881,E2 26488.881} C_VEL
LIN {X 0,Y 591.204,Z 340.396,A -85,B 0,C 180,E1 26488.293,E2 26488.293} C_VEL
LIN {X 0,Y 589.555,Z 337.457,A -85,B 0,C 180,E1 26487.911,E2 26487.911} C_VEL
LIN {X 0,Y 586.738,Z 335.031,A -85,B 0,C 180,E1 26487.34,E2 26487.34} C_VEL
LIN {X 0,Y 585.356,Z 331.986,A -85,B 0,C 180,E1 26486.984,E2 26486.984} C_VEL
LIN {X 0,Y 585.234,Z 331.272,A -85,B 0,C 180,E1 26486.921,E2 26486.921} C_VEL
LIN {X 0,Y 585.254,Z 331.289,A -85,B 0,C 180,E1 26483.565,E2 26483.565} C_VEL
LIN {X 0,Y 585.253,Z 331.312,A -85,B 0,C 180,E1 26480.289,E2 26480.289} C_VEL
LIN {X 0,Y 585.252,Z 331.31,A -85,B 0,C 180,E1 26476.987,E2 26476.987} C_VEL
LIN {X 0,Y 585.266,Z 331.347,A -85,B 0,C 180,E1 26474.421,E2 26474.421} C_VEL
LIN {X 0,Y 590.441,Z 347.93,A -85,B 0,C 180,E1 26473.665,E2 26473.665} C_VEL
LIN {X 0,Y 590.332,Z 429.486,A -85,B 0,C 180,E1 26470.802,E2 26470.802} C_VEL
LIN {X 0,Y 590.654,Z 510.012,A -85,B 0,C 180,E1 26467.832,E2 26467.832} C_VEL
LIN {X 0,Y 590.573,Z 585.574,A -85,B 0,C 180,E1 26464.954,E2 26464.954} C_VEL
LIN {X 0,Y 590,Z 663.403,A -85,B 0,C 180,E1 26461.894,E2 26461.894} C_VEL
LIN {X 0,Y 589.426,Z 724.729,A -85,B 0,C 180,E1 26459.465,E2 26459.465} C_VEL
LIN {X 0,Y 588.503,Z 802.993,A -85,B 0,C 180,E1 26456.298,E2 26456.298} C_VEL
LIN {X 0,Y 587.72,Z 848.985,A -85,B 0,C 180,E1 26454.424,E2 26454.424} C_VEL
LIN {X 0,Y 587.314,Z 855.326,A -85,B 0,C 180,E1 26454.2,E2 26454.2} C_VEL
LIN {X 0,Y 586.692,Z 969.277,A -85,B 0,C 180,E1 26452.724,E2 26452.724} C_VEL
LIN {X 0,Y 586.71,Z 981.563,A -85,B 0,C 180,E1 26452.438,E2 26452.438} C_VEL
LIN {X 0,Y 586.672,Z 993.42,A -85,B 0,C 180,E1 26452.038,E2 26452.038} C_VEL
LIN {X 0,Y 586.55,Z 1006.901,A -85,B 0,C 180,E1 26451.422,E2 26451.422} C_VEL
LIN {X 0,Y 586.332,Z 1018.871,A -85,B 0,C 180,E1 26450.677,E2 26450.677} C_VEL
LIN {X 0,Y 586.132,Z 1028.481,A -85,B 0,C 180,E1 26449.93,E2 26449.93} C_VEL
LIN {X 0,Y 585.927,Z 1036.447,A -85,B 0,C 180,E1 26449.18,E2 26449.18} C_VEL
LIN {X 0,Y 585.705,Z 1044.353,A -85,B 0,C 180,E1 26448.279,E2 26448.279} C_VEL
LIN {X 0,Y 585.496,Z 1051.508,A -85,B 0,C 180,E1 26447.273,E2 26447.273} C_VEL
LIN {X 0,Y 585.273,Z 1058.751,A -85,B 0,C 180,E1 26445.96,E2 26445.96} C_VEL
LIN {X 0,Y 585.121,Z 1063.55,A -85,B 0,C 180,E1 26444.742,E2 26444.742} C_VEL
LIN {X 0,Y 585.02,Z 1066.686,A -85,B 0,C 180,E1 26443.62,E2 26443.62} C_VEL
LIN {X 0,Y 584.961,Z 1068.658,A -85,B 0,C 180,E1 26442.492,E2 26442.492} C_VEL
LIN {X 0,Y 584.92,Z 1069.508,A -85,B 0,C 180,E1 26441.357,E2 26441.357} C_VEL
LIN {X 0,Y 584.915,Z 1069.157,A -85,B 0,C 180,E1 26440.087,E2 26440.087} C_VEL
LIN {X 0,Y 584.947,Z 1066.794,A -85,B 0,C 180,E1 26438.543,E2 26438.543} C_VEL
LIN {X 0,Y 585.016,Z 1063.509,A -85,B 0,C 180,E1 26437.362,E2 26437.362} C_VEL
LIN {X 0,Y 585.115,Z 1059.021,A -85,B 0,C 180,E1 26436.216,E2 26436.216} C_VEL
LIN {X 0,Y 585.282,Z 1052.953,A -85,B 0,C 180,E1 26435.041,E2 26435.041} C_VEL
LIN {X 0,Y 585.537,Z 1044.166,A -85,B 0,C 180,E1 26433.75,E2 26433.75} C_VEL
LIN {X 0,Y 585.769,Z 1035.678,A -85,B 0,C 180,E1 26432.776,E2 26432.776} C_VEL
LIN {X 0,Y 586.014,Z 1026.375,A -85,B 0,C 180,E1 26431.905,E2 26431.905} C_VEL
LIN {X 0,Y 586.271,Z 1014.814,A -85,B 0,C 180,E1 26431.029,E2 26431.029} C_VEL
LIN {X 0,Y 586.509,Z 1001.364,A -85,B 0,C 180,E1 26430.257,E2 26430.257} C_VEL
LIN {X 0,Y 586.649,Z 990.146,A -85,B 0,C 180,E1 26429.763,E2 26429.763} C_VEL
LIN {X 0,Y 586.732,Z 977.999,A -85,B 0,C 180,E1 26429.363,E2 26429.363} C_VEL
LIN {X 0,Y 586.757,Z 963.626,A -85,B 0,C 180,E1 26429.044,E2 26429.044} C_VEL
LIN {X 0,Y 587.49,Z 849.557,A -85,B 0,C 180,E1 26427.58,E2 26427.58} C_VEL
LIN {X 0,Y 587.567,Z 848.543,A -85,B 0,C 180,E1 26427.539,E2 26427.539} C_VEL
LIN {X 0,Y 587.224,Z 842.494,A -85,B 0,C 180,E1 26427.273,E2 26427.273} C_VEL
LIN {X 0,Y 584.341,Z 832.92,A -85,B 0,C 180,E1 26426.786,E2 26426.786} C_VEL
LIN {X 0,Y 581.014,Z 822.38,A -85,B 0,C 180,E1 26426.242,E2 26426.242} C_VEL
LIN {X 0,Y 580.535,Z 817.332,A -85,B 0,C 180,E1 26426.012,E2 26426.012} C_VEL
LIN {X 0,Y 581.909,Z 735.659,A -85,B 0,C 180,E1 26422.548,E2 26422.548} C_VEL
LIN {X 0,Y 583.027,Z 677.37,A -85,B 0,C 180,E1 26420.053,E2 26420.053} C_VEL
LIN {X 0,Y 584.211,Z 678.898,A -85,B 0,C 180,E1 26419.88,E2 26419.88} C_VEL
LIN {X 0,Y 586.069,Z 678.582,A -85,B 0,C 180,E1 26419.681,E2 26419.681} C_VEL
LIN {X 0,Y 589.016,Z 675.686,A -85,B 0,C 180,E1 26419.43,E2 26419.43} C_VEL
LIN {X 0,Y 592.682,Z 669.871,A -85,B 0,C 180,E1 26419.176,E2 26419.176} C_VEL
LIN {X 0,Y 596.077,Z 668.392,A -85,B 0,C 180,E1 26418.854,E2 26418.854} C_VEL
LIN {X 0,Y 599.972,Z 664.609,A -85,B 0,C 180,E1 26418.544,E2 26418.544} C_VEL
LIN {X 0,Y 603.114,Z 660.169,A -85,B 0,C 180,E1 26418.332,E2 26418.332} C_VEL
LIN {X 0,Y 607.776,Z 657.362,A -85,B 0,C 180,E1 26417.965,E2 26417.965} C_VEL
LIN {X 0,Y 612.66,Z 652.272,A -85,B 0,C 180,E1 26417.636,E2 26417.636} C_VEL
LIN {X 0,Y 614.453,Z 650.24,A -85,B 0,C 180,E1 26417.52,E2 26417.52} C_VEL
LIN {X 0,Y 619.851,Z 646.474,A -85,B 0,C 180,E1 26417.13,E2 26417.13} C_VEL
LIN {X 0,Y 620.331,Z 646.144,A -85,B 0,C 180,E1 26417.095,E2 26417.095} C_VEL
LIN {X 0,Y 616.972,Z 766.217,A -85,B 0,C 180,E1 26415.379,E2 26415.379} C_VEL
LIN {X 0,Y 615.721,Z 809.824,A -85,B 0,C 180,E1 26414.756,E2 26414.756} C_VEL
LIN {X 0,Y 614.29,Z 836.155,A -85,B 0,C 180,E1 26414.213,E2 26414.213} C_VEL
LIN {X 0,Y 612.796,Z 858.535,A -85,B 0,C 180,E1 26413.629,E2 26413.629} C_VEL
LIN {X 0,Y 611.04,Z 881.488,A -85,B 0,C 180,E1 26412.902,E2 26412.902} C_VEL
LIN {X 0,Y 608.576,Z 909.082,A -85,B 0,C 180,E1 26411.841,E2 26411.841} C_VEL
LIN {X 0,Y 606.288,Z 929.004,A -85,B 0,C 180,E1 26410.9,E2 26410.9} C_VEL
LIN {X 0,Y 603.515,Z 949.631,A -85,B 0,C 180,E1 26409.756,E2 26409.756} C_VEL
LIN {X 0,Y 600.787,Z 968.864,A -85,B 0,C 180,E1 26408.551,E2 26408.551} C_VEL
LIN {X 0,Y 598.057,Z 987.419,A -85,B 0,C 180,E1 26407.246,E2 26407.246} C_VEL
LIN {X 0,Y 595.288,Z 1005.767,A -85,B 0,C 180,E1 26405.805,E2 26405.805} C_VEL
LIN {X 0,Y 592.5,Z 1024.151,A -85,B 0,C 180,E1 26404.192,E2 26404.192} C_VEL
LIN {X 0,Y 589.259,Z 1045.522,A -85,B 0,C 180,E1 26402.082,E2 26402.082} C_VEL
LIN {X 0,Y 586.446,Z 1064.144,A -85,B 0,C 180,E1 26399.972,E2 26399.972} C_VEL
LIN {X 0,Y 584.33,Z 1079.154,A -85,B 0,C 180,E1 26398.072,E2 26398.072} C_VEL
LIN {X 0,Y 582.439,Z 1093.044,A -85,B 0,C 180,E1 26396.123,E2 26396.123} C_VEL
LIN {X 0,Y 580.668,Z 1107.398,A -85,B 0,C 180,E1 26393.871,E2 26393.871} C_VEL
LIN {X 0,Y 578.998,Z 1122.412,A -85,B 0,C 180,E1 26391.158,E2 26391.158} C_VEL
LIN {X 0,Y 578.02,Z 1132.459,A -85,B 0,C 180,E1 26389.084,E2 26389.084} C_VEL
LIN {X 0,Y 577.285,Z 1141.295,A -85,B 0,C 180,E1 26387.022,E2 26387.022} C_VEL
LIN {X 0,Y 576.756,Z 1149.345,A -85,B 0,C 180,E1 26384.868,E2 26384.868} C_VEL
LIN {X 0,Y 576.373,Z 1156.233,A -85,B 0,C 180,E1 26382.729,E2 26382.729} C_VEL
LIN {X 0,Y 576.129,Z 1162.462,A -85,B 0,C 180,E1 26380.4,E2 26380.4} C_VEL
LIN {X 0,Y 575.996,Z 1167.596,A -85,B 0,C 180,E1 26377.984,E2 26377.984} C_VEL
LIN {X 0,Y 575.927,Z 1171.886,A -85,B 0,C 180,E1 26375.181,E2 26375.181} C_VEL
LIN {X 0,Y 575.908,Z 1174.161,A -85,B 0,C 180,E1 26372.588,E2 26372.588} C_VEL
LIN {X 0,Y 575.901,Z 1174.925,A -85,B 0,C 180,E1 26370.2,E2 26370.2} C_VEL
LIN {X 0,Y 575.91,Z 1174.352,A -85,B 0,C 180,E1 26367.713,E2 26367.713} C_VEL
LIN {X 0,Y 575.915,Z 1172.586,A -85,B 0,C 180,E1 26365.421,E2 26365.421} C_VEL
LIN {X 0,Y 575.95,Z 1169.465,A -85,B 0,C 180,E1 26363.021,E2 26363.021} C_VEL
LIN {X 0,Y 576.07,Z 1164.37,A -85,B 0,C 180,E1 26360.309,E2 26360.309} C_VEL
LIN {X 0,Y 576.306,Z 1157.58,A -85,B 0,C 180,E1 26357.637,E2 26357.637} C_VEL
LIN {X 0,Y 576.682,Z 1150.37,A -85,B 0,C 180,E1 26355.338,E2 26355.338} C_VEL
LIN {X 0,Y 577.201,Z 1142.472,A -85,B 0,C 180,E1 26353.186,E2 26353.186} C_VEL
LIN {X 0,Y 577.902,Z 1133.795,A -85,B 0,C 180,E1 26351.124,E2 26351.124} C_VEL
LIN {X 0,Y 578.779,Z 1124.43,A -85,B 0,C 180,E1 26349.154,E2 26349.154} C_VEL
LIN {X 0,Y 579.897,Z 1113.909,A -85,B 0,C 180,E1 26347.174,E2 26347.174} C_VEL
LIN {X 0,Y 581.285,Z 1102.124,A -85,B 0,C 180,E1 26345.185,E2 26345.185} C_VEL
LIN {X 0,Y 583.318,Z 1086.501,A -85,B 0,C 180,E1 26342.829,E2 26342.829} C_VEL
LIN {X 0,Y 585.869,Z 1068.35,A -85,B 0,C 180,E1 26340.449,E2 26340.449} C_VEL
LIN {X 0,Y 588.244,Z 1052.052,A -85,B 0,C 180,E1 26338.547,E2 26338.547} C_VEL
LIN {X 0,Y 590.826,Z 1034.913,A -85,B 0,C 180,E1 26336.75,E2 26336.75} C_VEL
LIN {X 0,Y 594.057,Z 1014.05,A -85,B 0,C 180,E1 26334.799,E2 26334.799} C_VEL
LIN {X 0,Y 597.493,Z 991.322,A -85,B 0,C 180,E1 26332.956,E2 26332.956} C_VEL
LIN {X 0,Y 600.292,Z 972.313,A -85,B 0,C 180,E1 26331.591,E2 26331.591} C_VEL
LIN {X 0,Y 602.85,Z 954.404,A -85,B 0,C 180,E1 26330.441,E2 26330.441} C_VEL
LIN {X 0,Y 605.312,Z 936.268,A -85,B 0,C 180,E1 26329.398,E2 26329.398} C_VEL
LIN {X 0,Y 607.524,Z 918.547,A -85,B 0,C 180,E1 26328.492,E2 26328.492} C_VEL
LIN {X 0,Y 609.45,Z 899.2,A -85,B 0,C 180,E1 26327.666,E2 26327.666} C_VEL
LIN {X 0,Y 611.348,Z 877.447,A -85,B 0,C 180,E1 26326.872,E2 26326.872} C_VEL
LIN {X 0,Y 612.967,Z 856.151,A -85,B 0,C 180,E1 26326.214,E2 26326.214} C_VEL
LIN {X 0,Y 614.445,Z 833.729,A -85,B 0,C 180,E1 26325.641,E2 26325.641} C_VEL
LIN {X 0,Y 615.909,Z 804.912,A -85,B 0,C 180,E1 26325.076,E2 26325.076} C_VEL
LIN {X 0,Y 619.684,Z 665.748,A -85,B 0,C 180,E1 26323.105,E2 26323.105} C_VEL
LIN {X 0,Y 628.471,Z 431.256,A -85,B 0,C 180,E1 26319.576,E2 26319.576} C_VEL
LIN {X 0,Y 629.487,Z 401.051,A -85,B 0,C 180,E1 26319.132,E2 26319.132} C_VEL
LIN {X 0,Y 616.675,Z 388.439,A -85,B 0,C 180,E1 26317.389,E2 26317.389} C_VEL
LIN {X 0,Y 608.094,Z 380.525,A -85,B 0,C 180,E1 26316.15,E2 26316.15} C_VEL
LIN {X 0,Y 602.483,Z 375.132,A -85,B 0,C 180,E1 26315.264,E2 26315.264} C_VEL
LIN {X 0,Y 599.375,Z 369.729,A -85,B 0,C 180,E1 26313.517,E2 26313.517} C_VEL
LIN {X 0,Y 596.753,Z 364.924,A -85,B 0,C 180,E1 26311.846,E2 26311.846} C_VEL
LIN {X 0,Y 594.505,Z 360.967,A -85,B 0,C 180,E1 26310.303,E2 26310.303} C_VEL
LIN {X 0,Y 593.621,Z 359.549,A -85,B 0,C 180,E1 26309.684,E2 26309.684} C_VEL
LIN {X 0,Y 591.424,Z 355.639,A -85,B 0,C 180,E1 26307.925,E2 26307.925} C_VEL
LIN {X 0,Y 590.839,Z 354.562,A -85,B 0,C 180,E1 26307.407,E2 26307.407} C_VEL
LIN {X 0,Y 588.401,Z 350.899,A -85,B 0,C 180,E1 26305.248,E2 26305.248} C_VEL
LIN {X 0,Y 587.82,Z 349.276,A -85,B 0,C 180,E1 26304.415,E2 26304.415} C_VEL
LIN {X 0,Y 584.887,Z 344.856,A -85,B 0,C 180,E1 26300.62,E2 26300.62} C_VEL
LIN {X 0,Y 584.422,Z 343.684,A -85,B 0,C 180,E1 26299.489,E2 26299.489} C_VEL
LIN {X 0,Y 582.843,Z 342.208,A -85,B 0,C 180,E1 26294.912,E2 26294.912} C_VEL
LIN {X 0,Y 583.34,Z 342.757,A -85,B 0,C 180,E1 26290.968,E2 26290.968} C_VEL
LIN {X 0,Y 584.758,Z 344.255,A -85,B 0,C 180,E1 26288.107,E2 26288.107} C_VEL
LIN {X 0,Y 587.785,Z 349.277,A -85,B 0,C 180,E1 26283.902,E2 26283.902} C_VEL
LIN {X 0,Y 588.345,Z 350.485,A -85,B 0,C 180,E1 26283.215,E2 26283.215} C_VEL
LIN {X 0,Y 590.622,Z 354.335,A -85,B 0,C 180,E1 26281.067,E2 26281.067} C_VEL
LIN {X 0,Y 591.432,Z 355.313,A -85,B 0,C 180,E1 26280.484,E2 26280.484} C_VEL
LIN {X 0,Y 593.359,Z 359.193,A -85,B 0,C 180,E1 26278.841,E2 26278.841} C_VEL
LIN {X 0,Y 594.593,Z 360.766,A -85,B 0,C 180,E1 26278.073,E2 26278.073} C_VEL
LIN {X 0,Y 596.791,Z 364.844,A -85,B 0,C 180,E1 26276.542,E2 26276.542} C_VEL
LIN {X 0,Y 597.709,Z 366.399,A -85,B 0,C 180,E1 26275.971,E2 26275.971} C_VEL
LIN {X 0,Y 600.591,Z 371.426,A -85,B 0,C 180,E1 26274.267,E2 26274.267} C_VEL
LIN {X 0,Y 603.466,Z 376.702,A -85,B 0,C 180,E1 26272.67,E2 26272.67} C_VEL
LIN {X 0,Y 606.368,Z 382.035,A -85,B 0,C 180,E1 26271.179,E2 26271.179} C_VEL
LIN {X 0,Y 609.422,Z 387.779,A -85,B 0,C 180,E1 26269.698,E2 26269.698} C_VEL
LIN {X 0,Y 613.712,Z 395.854,A -85,B 0,C 180,E1 26267.772,E2 26267.772} C_VEL
LIN {X 0,Y 619.985,Z 408.278,A -85,B 0,C 180,E1 26265.142,E2 26265.142} C_VEL
LIN {X 0,Y 626.39,Z 421.717,A -85,B 0,C 180,E1 26262.632,E2 26262.632} C_VEL
LIN {X 0,Y 627.073,Z 423.731,A -85,B 0,C 180,E1 26262.316,E2 26262.316} C_VEL
LIN {X 0,Y 622.89,Z 456.298,A -85,B 0,C 180,E1 26259.57,E2 26259.57} C_VEL
LIN {X 0,Y 618.623,Z 491.636,A -85,B 0,C 180,E1 26256.722,E2 26256.722} C_VEL
LIN {X 0,Y 614.4,Z 528.997,A -85,B 0,C 180,E1 26253.83,E2 26253.83} C_VEL
LIN {X 0,Y 609.301,Z 583.268,A -85,B 0,C 180,E1 26249.748,E2 26249.748} C_VEL
LIN {X 0,Y 609.76,Z 600.011,A -85,B 0,C 180,E1 26248.349,E2 26248.349} C_VEL
LIN {X 0,Y 612.128,Z 615.258,A -85,B 0,C 180,E1 26246.936,E2 26246.936} C_VEL
LIN {X 0,Y 616.607,Z 629.586,A -85,B 0,C 180,E1 26245.461,E2 26245.461} C_VEL
LIN {X 0,Y 622.556,Z 641.408,A -85,B 0,C 180,E1 26244.11,E2 26244.11} C_VEL
LIN {X 0,Y 630.054,Z 651.835,A -85,B 0,C 180,E1 26242.797,E2 26242.797} C_VEL
LIN {X 0,Y 639.864,Z 661.556,A -85,B 0,C 180,E1 26241.427,E2 26241.427} C_VEL
LIN {X 0,Y 650.926,Z 669.42,A -85,B 0,C 180,E1 26240.166,E2 26240.166} C_VEL
LIN {X 0,Y 662.383,Z 675.315,A -85,B 0,C 180,E1 26239.07,E2 26239.07} C_VEL
LIN {X 0,Y 675.153,Z 680.011,A -85,B 0,C 180,E1 26238.024,E2 26238.024} C_VEL
LIN {X 0,Y 657.446,Z 700.927,A -85,B 0,C 180,E1 26237.721,E2 26237.721} C_VEL
LIN {X 0,Y 648.737,Z 712.988,A -85,B 0,C 180,E1 26237.451,E2 26237.451} C_VEL
LIN {X 0,Y 644.564,Z 719.628,A -85,B 0,C 180,E1 26237.264,E2 26237.264} C_VEL
LIN {X 0,Y 635.729,Z 731.597,A -85,B 0,C 180,E1 26236.998,E2 26236.998} C_VEL
LIN {X 0,Y 629.062,Z 742.812,A -85,B 0,C 180,E1 26236.649,E2 26236.649} C_VEL
LIN {X 0,Y 621.123,Z 758.329,A -85,B 0,C 180,E1 26236.103,E2 26236.103} C_VEL
LIN {X 0,Y 619.869,Z 771.553,A -85,B 0,C 180,E1 26236.011,E2 26236.011} C_VEL
LIN {X 0,Y 618.349,Z 824.299,A -85,B 0,C 180,E1 26235.268,E2 26235.268} C_VEL
LIN {X 0,Y 616.625,Z 852.604,A -85,B 0,C 180,E1 26234.737,E2 26234.737} C_VEL
LIN {X 0,Y 614.548,Z 879.633,A -85,B 0,C 180,E1 26234.061,E2 26234.061} C_VEL
LIN {X 0,Y 612.258,Z 905.377,A -85,B 0,C 180,E1 26233.25,E2 26233.25} C_VEL
LIN {X 0,Y 609.595,Z 931.005,A -85,B 0,C 180,E1 26232.258,E2 26232.258} C_VEL
LIN {X 0,Y 606.7,Z 955.797,A -85,B 0,C 180,E1 26231.114,E2 26231.114} C_VEL
LIN {X 0,Y 603.573,Z 979.625,A -85,B 0,C 180,E1 26229.811,E2 26229.811} C_VEL
LIN {X 0,Y 600.272,Z 1002.703,A -85,B 0,C 180,E1 26228.343,E2 26228.343} C_VEL
LIN {X 0,Y 596.836,Z 1025.703,A -85,B 0,C 180,E1 26226.665,E2 26226.665} C_VEL
LIN {X 0,Y 593.372,Z 1048.279,A -85,B 0,C 180,E1 26224.776,E2 26224.776} C_VEL
LIN {X 0,Y 590.215,Z 1069.352,A -85,B 0,C 180,E1 26222.768,E2 26222.768} C_VEL
LIN {X 0,Y 587.335,Z 1088.26,A -85,B 0,C 180,E1 26220.71,E2 26220.71} C_VEL
LIN {X 0,Y 584.701,Z 1106.509,A -85,B 0,C 180,E1 26218.479,E2 26218.479} C_VEL
LIN {X 0,Y 582.547,Z 1122.283,A -85,B 0,C 180,E1 26216.283,E2 26216.283} C_VEL
LIN {X 0,Y 580.644,Z 1137.722,A -85,B 0,C 180,E1 26213.869,E2 26213.869} C_VEL
LIN {X 0,Y 579.045,Z 1152.194,A -85,B 0,C 180,E1 26211.26,E2 26211.26} C_VEL
LIN {X 0,Y 577.896,Z 1164.112,A -85,B 0,C 180,E1 26208.772,E2 26208.772} C_VEL
LIN {X 0,Y 577.054,Z 1174.748,A -85,B 0,C 180,E1 26206.197,E2 26206.197} C_VEL
LIN {X 0,Y 576.485,Z 1184.275,A -85,B 0,C 180,E1 26203.438,E2 26203.438} C_VEL
LIN {X 0,Y 576.146,Z 1191.668,A -85,B 0,C 180,E1 26200.8,E2 26200.8} C_VEL
LIN {X 0,Y 575.995,Z 1197.328,A -85,B 0,C 180,E1 26198.182,E2 26198.182} C_VEL
LIN {X 0,Y 575.932,Z 1201.411,A -85,B 0,C 180,E1 26195.578,E2 26195.578} C_VEL
LIN {X 0,Y 575.916,Z 1203.979,A -85,B 0,C 180,E1 26192.984,E2 26192.984} C_VEL
LIN {X 0,Y 575.893,Z 1204.916,A -85,B 0,C 180,E1 26190.496,E2 26190.496} C_VEL
LIN {X 0,Y 575.911,Z 1204.464,A -85,B 0,C 180,E1 26187.909,E2 26187.909} C_VEL
LIN {X 0,Y 575.916,Z 1202.599,A -85,B 0,C 180,E1 26185.418,E2 26185.418} C_VEL
LIN {X 0,Y 575.966,Z 1199.087,A -85,B 0,C 180,E1 26182.818,E2 26182.818} C_VEL
LIN {X 0,Y 576.083,Z 1193.783,A -85,B 0,C 180,E1 26180.105,E2 26180.105} C_VEL
LIN {X 0,Y 576.333,Z 1187.029,A -85,B 0,C 180,E1 26177.474,E2 26177.474} C_VEL
LIN {X 0,Y 576.791,Z 1178.839,A -85,B 0,C 180,E1 26174.925,E2 26174.925} C_VEL
LIN {X 0,Y 577.483,Z 1169.009,A -85,B 0,C 180,E1 26172.361,E2 26172.361} C_VEL
LIN {X 0,Y 578.554,Z 1156.841,A -85,B 0,C 180,E1 26169.672,E2 26169.672} C_VEL
LIN {X 0,Y 579.877,Z 1144.328,A -85,B 0,C 180,E1 26167.278,E2 26167.278} C_VEL
LIN {X 0,Y 581.59,Z 1129.896,A -85,B 0,C 180,E1 26164.871,E2 26164.871} C_VEL
LIN {X 0,Y 583.838,Z 1112.618,A -85,B 0,C 180,E1 26162.346,E2 26162.346} C_VEL
LIN {X 0,Y 586.172,Z 1096.3,A -85,B 0,C 180,E1 26160.238,E2 26160.238} C_VEL
LIN {X 0,Y 589.025,Z 1076.825,A -85,B 0,C 180,E1 26158.019,E2 26158.019} C_VEL
LIN {X 0,Y 592.01,Z 1057.493,A -85,B 0,C 180,E1 26156.067,E2 26156.067} C_VEL
LIN {X 0,Y 595.273,Z 1036.059,A -85,B 0,C 180,E1 26154.169,E2 26154.169} C_VEL
LIN {X 0,Y 598.71,Z 1013.017,A -85,B 0,C 180,E1 26152.38,E2 26152.38} C_VEL
LIN {X 0,Y 602.11,Z 989.79,A -85,B 0,C 180,E1 26150.811,E2 26150.811} C_VEL
LIN {X 0,Y 605.446,Z 965.746,A -85,B 0,C 180,E1 26149.406,E2 26149.406} C_VEL
LIN {X 0,Y 608.15,Z 943.868,A -85,B 0,C 180,E1 26148.312,E2 26148.312} C_VEL
LIN {X 0,Y 610.968,Z 918.103,A -85,B 0,C 180,E1 26147.22,E2 26147.22} C_VEL
LIN {X 0,Y 613.595,Z 890.829,A -85,B 0,C 180,E1 26146.271,E2 26146.271} C_VEL
LIN {X 0,Y 615.881,Z 863.099,A -85,B 0,C 180,E1 26145.504,E2 26145.504} C_VEL
LIN {X 0,Y 617.78,Z 835.071,A -85,B 0,C 180,E1 26144.912,E2 26144.912} C_VEL
LIN {X 0,Y 619.117,Z 803.748,A -85,B 0,C 180,E1 26144.428,E2 26144.428} C_VEL
LIN {X 0,Y 620.726,Z 747.175,A -85,B 0,C 180,E1 26143.645,E2 26143.645} C_VEL
LIN {X 0,Y 628.018,Z 660.316,A -85,B 0,C 180,E1 26142.188,E2 26142.188} C_VEL
LIN {X 0,Y 629.413,Z 644.875,A -85,B 0,C 180,E1 26141.938,E2 26141.938} C_VEL
LIN {X 0,Y 632.515,Z 611.144,A -85,B 0,C 180,E1 26141.396,E2 26141.396} C_VEL
LIN {X 0,Y 634.272,Z 594.59,A -85,B 0,C 180,E1 26141.153,E2 26141.153} C_VEL
LIN {X 0,Y 636.597,Z 566.988,A -85,B 0,C 180,E1 26140.69,E2 26140.69} C_VEL
LIN {X 0,Y 640.139,Z 536.711,A -85,B 0,C 180,E1 26140.278,E2 26140.278} C_VEL
LIN {X 0,Y 642.014,Z 512.84,A -85,B 0,C 180,E1 26139.863,E2 26139.863} C_VEL
LIN {X 0,Y 646.2,Z 479.543,A -85,B 0,C 180,E1 26139.441,E2 26139.441} C_VEL
LIN {X 0,Y 646.854,Z 473.301,A -85,B 0,C 180,E1 26139.35,E2 26139.35} C_VEL
LIN {X 0,Y 648.348,Z 452.706,A -85,B 0,C 180,E1 26138.979,E2 26138.979} C_VEL
LIN {X 0,Y 650.884,Z 430.557,A -85,B 0,C 180,E1 26138.674,E2 26138.674} C_VEL
LIN {X 0,Y 639.891,Z 418.919,A -85,B 0,C 180,E1 26137.209,E2 26137.209} C_VEL
LIN {X 0,Y 621.488,Z 391.777,A -85,B 0,C 180,E1 26134.299,E2 26134.299} C_VEL
LIN {X 0,Y 610.674,Z 376.63,A -85,B 0,C 180,E1 26132.428,E2 26132.428} C_VEL
LIN {X 0,Y 602.669,Z 365.864,A -85,B 0,C 180,E1 26130.952,E2 26130.952} C_VEL
LIN {X 0,Y 598.782,Z 360.709,A -85,B 0,C 180,E1 26130.202,E2 26130.202} C_VEL
LIN {X 0,Y 594.867,Z 355.567,A -85,B 0,C 180,E1 26129.422,E2 26129.422} C_VEL
LIN {X 0,Y 591.581,Z 351.164,A -85,B 0,C 180,E1 26128.742,E2 26128.742} C_VEL
LIN {X 0,Y 587.761,Z 346.706,A -85,B 0,C 180,E1 26127.949,E2 26127.949} C_VEL
LIN {X 0,Y 586.383,Z 344.515,A -85,B 0,C 180,E1 26127.633,E2 26127.633} C_VEL
LIN {X 0,Y 583.349,Z 341.381,A -85,B 0,C 180,E1 26126.988,E2 26126.988} C_VEL
LIN {X 0,Y 581.784,Z 338.482,A -85,B 0,C 180,E1 26126.597,E2 26126.597} C_VEL
LIN {X 0,Y 578.863,Z 336.081,A -85,B 0,C 180,E1 26125.969,E2 26125.969} C_VEL
LIN {X 0,Y 577.439,Z 333.115,A -85,B 0,C 180,E1 26125.583,E2 26125.583} C_VEL
LIN {X 0,Y 577.278,Z 332.237,A -85,B 0,C 180,E1 26125.501,E2 26125.501} C_VEL
LIN {X 0,Y 577.312,Z 332.324,A -85,B 0,C 180,E1 26122.291,E2 26122.291} C_VEL
LIN {X 0,Y 577.289,Z 332.323,A -85,B 0,C 180,E1 26119.109,E2 26119.109} C_VEL
LIN {X 0,Y 577.319,Z 332.315,A -85,B 0,C 180,E1 26115.778,E2 26115.778} C_VEL
LIN {X 0,Y 577.317,Z 332.441,A -85,B 0,C 180,E1 26114.692,E2 26114.692} C_VEL
LIN {X 0,Y 582.899,Z 349.899,A -85,B 0,C 180,E1 26113.873,E2 26113.873} C_VEL
LIN {X 0,Y 582.77,Z 427.165,A -85,B 0,C 180,E1 26111.154,E2 26111.154} C_VEL
LIN {X 0,Y 583.046,Z 507.587,A -85,B 0,C 180,E1 26108.183,E2 26108.183} C_VEL
LIN {X 0,Y 582.964,Z 580.151,A -85,B 0,C 180,E1 26105.413,E2 26105.413} C_VEL
LIN {X 0,Y 582.45,Z 655.518,A -85,B 0,C 180,E1 26102.46,E2 26102.46} C_VEL
LIN {X 0,Y 581.611,Z 736.858,A -85,B 0,C 180,E1 26099.212,E2 26099.212} C_VEL
LIN {X 0,Y 580.614,Z 816.719,A -85,B 0,C 180,E1 26095.951,E2 26095.951} C_VEL
LIN {X 0,Y 579.956,Z 849.542,A -85,B 0,C 180,E1 26094.608,E2 26094.608} C_VEL
LIN {X 0,Y 579.507,Z 856.491,A -85,B 0,C 180,E1 26094.361,E2 26094.361} C_VEL
LIN {X 0,Y 578.848,Z 970.384,A -85,B 0,C 180,E1 26092.859,E2 26092.859} C_VEL
LIN {X 0,Y 578.872,Z 982.811,A -85,B 0,C 180,E1 26092.566,E2 26092.566} C_VEL
LIN {X 0,Y 578.834,Z 994.759,A -85,B 0,C 180,E1 26092.157,E2 26092.157} C_VEL
LIN {X 0,Y 578.712,Z 1007.785,A -85,B 0,C 180,E1 26091.555,E2 26091.555} C_VEL
LIN {X 0,Y 578.489,Z 1019.845,A -85,B 0,C 180,E1 26090.8,E2 26090.8} C_VEL
LIN {X 0,Y 578.279,Z 1029.498,A -85,B 0,C 180,E1 26090.043,E2 26090.043} C_VEL
LIN {X 0,Y 578.051,Z 1037.977,A -85,B 0,C 180,E1 26089.233,E2 26089.233} C_VEL
LIN {X 0,Y 577.83,Z 1045.53,A -85,B 0,C 180,E1 26088.357,E2 26088.357} C_VEL
LIN {X 0,Y 577.621,Z 1052.275,A -85,B 0,C 180,E1 26087.402,E2 26087.402} C_VEL
LIN {X 0,Y 577.405,Z 1059.167,A -85,B 0,C 180,E1 26086.174,E2 26086.174} C_VEL
LIN {X 0,Y 577.218,Z 1064.517,A -85,B 0,C 180,E1 26084.837,E2 26084.837} C_VEL
LIN {X 0,Y 577.109,Z 1067.701,A -85,B 0,C 180,E1 26083.699,E2 26083.699} C_VEL
LIN {X 0,Y 577.042,Z 1069.715,A -85,B 0,C 180,E1 26082.556,E2 26082.556} C_VEL
LIN {X 0,Y 576.998,Z 1070.6,A -85,B 0,C 180,E1 26081.406,E2 26081.406} C_VEL
LIN {X 0,Y 576.987,Z 1070.34,A -85,B 0,C 180,E1 26080.22,E2 26080.22} C_VEL
LIN {X 0,Y 577.018,Z 1068.468,A -85,B 0,C 180,E1 26078.767,E2 26078.767} C_VEL
LIN {X 0,Y 577.096,Z 1064.777,A -85,B 0,C 180,E1 26077.378,E2 26077.378} C_VEL
LIN {X 0,Y 577.193,Z 1060.716,A -85,B 0,C 180,E1 26076.303,E2 26076.303} C_VEL
LIN {X 0,Y 577.338,Z 1055.392,A -85,B 0,C 180,E1 26075.221,E2 26075.221} C_VEL
LIN {X 0,Y 577.541,Z 1048.622,A -85,B 0,C 180,E1 26074.133,E2 26074.133} C_VEL
LIN {X 0,Y 577.835,Z 1039.12,A -85,B 0,C 180,E1 26072.929,E2 26072.929} C_VEL
LIN {X 0,Y 578.112,Z 1029.003,A -85,B 0,C 180,E1 26071.937,E2 26071.937} C_VEL
LIN {X 0,Y 578.342,Z 1019.282,A -85,B 0,C 180,E1 26071.16,E2 26071.16} C_VEL
LIN {X 0,Y 578.579,Z 1008.451,A -85,B 0,C 180,E1 26070.458,E2 26070.458} C_VEL
LIN {X 0,Y 578.803,Z 994.621,A -85,B 0,C 180,E1 26069.763,E2 26069.763} C_VEL
LIN {X 0,Y 578.896,Z 981.087,A -85,B 0,C 180,E1 26069.284,E2 26069.284} C_VEL
LIN {X 0,Y 578.924,Z 968.82,A -85,B 0,C 180,E1 26068.983,E2 26068.983} C_VEL
LIN {X 0,Y 578.914,Z 946.679,A -85,B 0,C 180,E1 26068.666,E2 26068.666} C_VEL
LIN {X 0,Y 579.694,Z 850.579,A -85,B 0,C 180,E1 26067.412,E2 26067.412} C_VEL
LIN {X 0,Y 580.337,Z 829.778,A -85,B 0,C 180,E1 26066.541,E2 26066.541} C_VEL
LIN {X 0,Y 580.535,Z 817.332,A -85,B 0,C 180,E1 26066.012,E2 26066.012} C_VEL
LIN {X 0,Y 579.683,Z 810.344,A -85,B 0,C 180,E1 26065.689,E2 26065.689} C_VEL
LIN {X 0,Y 573.976,Z 792.244,A -85,B 0,C 180,E1 26064.738,E2 26064.738} C_VEL
LIN {X 0,Y 573.35,Z 786.217,A -85,B 0,C 180,E1 26064.461,E2 26064.461} C_VEL
LIN {X 0,Y 574.855,Z 704.699,A -85,B 0,C 180,E1 26060.975,E2 26060.975} C_VEL
LIN {X 0,Y 575.112,Z 694.453,A -85,B 0,C 180,E1 26060.517,E2 26060.517} C_VEL
LIN {X 0,Y 576.078,Z 695.848,A -85,B 0,C 180,E1 26060.367,E2 26060.367} C_VEL
LIN {X 0,Y 577.71,Z 695.789,A -85,B 0,C 180,E1 26060.179,E2 26060.179} C_VEL
LIN {X 0,Y 580.4,Z 693.5,A -85,B 0,C 180,E1 26059.934,E2 26059.934} C_VEL
LIN {X 0,Y 584.079,Z 687.837,A -85,B 0,C 180,E1 26059.668,E2 26059.668} C_VEL
LIN {X 0,Y 584.838,Z 686.778,A -85,B 0,C 180,E1 26059.611,E2 26059.611} C_VEL
LIN {X 0,Y 588.217,Z 685.193,A -85,B 0,C 180,E1 26059.283,E2 26059.283} C_VEL
LIN {X 0,Y 592.085,Z 681.324,A -85,B 0,C 180,E1 26058.966,E2 26058.966} C_VEL
LIN {X 0,Y 595.203,Z 676.856,A -85,B 0,C 180,E1 26058.748,E2 26058.748} C_VEL
LIN {X 0,Y 599.718,Z 673.9,A -85,B 0,C 180,E1 26058.363,E2 26058.363} C_VEL
LIN {X 0,Y 604.417,Z 668.811,A -85,B 0,C 180,E1 26058.029,E2 26058.029} C_VEL
LIN {X 0,Y 606.135,Z 666.718,A -85,B 0,C 180,E1 26057.921,E2 26057.921} C_VEL
LIN {X 0,Y 611.613,Z 662.909,A -85,B 0,C 180,E1 26057.531,E2 26057.531} C_VEL
LIN {X 0,Y 613.886,Z 660.889,A -85,B 0,C 180,E1 26057.376,E2 26057.376} C_VEL
LIN {X 0,Y 610.398,Z 769.756,A -85,B 0,C 180,E1 26055.77,E2 26055.77} C_VEL
LIN {X 0,Y 608.837,Z 813.769,A -85,B 0,C 180,E1 26055.099,E2 26055.099} C_VEL
LIN {X 0,Y 607.408,Z 839.561,A -85,B 0,C 180,E1 26054.551,E2 26054.551} C_VEL
LIN {X 0,Y 605.617,Z 866.077,A -85,B 0,C 180,E1 26053.835,E2 26053.835} C_VEL
LIN {X 0,Y 603.351,Z 892.131,A -85,B 0,C 180,E1 26052.932,E2 26052.932} C_VEL
LIN {X 0,Y 601.165,Z 914.502,A -85,B 0,C 180,E1 26052.013,E2 26052.013} C_VEL
LIN {X 0,Y 598.974,Z 934.559,A -85,B 0,C 180,E1 26051.063,E2 26051.063} C_VEL
LIN {X 0,Y 597.168,Z 949.531,A -85,B 0,C 180,E1 26050.265,E2 26050.265} C_VEL
LIN {X 0,Y 594.446,Z 968.011,A -85,B 0,C 180,E1 26049.108,E2 26049.108} C_VEL
LIN {X 0,Y 591.554,Z 986.717,A -85,B 0,C 180,E1 26047.788,E2 26047.788} C_VEL
LIN {X 0,Y 588.664,Z 1004.863,A -85,B 0,C 180,E1 26046.357,E2 26046.357} C_VEL
LIN {X 0,Y 585.857,Z 1022.337,A -85,B 0,C 180,E1 26044.822,E2 26044.822} C_VEL
LIN {X 0,Y 582.972,Z 1040.391,A -85,B 0,C 180,E1 26043.054,E2 26043.054} C_VEL
LIN {X 0,Y 579.603,Z 1061.531,A -85,B 0,C 180,E1 26040.707,E2 26040.707} C_VEL
LIN {X 0,Y 577.141,Z 1077.573,A -85,B 0,C 180,E1 26038.68,E2 26038.68} C_VEL
LIN {X 0,Y 575.183,Z 1091.226,A -85,B 0,C 180,E1 26036.76,E2 26036.76} C_VEL
LIN {X 0,Y 573.501,Z 1103.519,A -85,B 0,C 180,E1 26034.847,E2 26034.847} C_VEL
LIN {X 0,Y 572.06,Z 1115.158,A -85,B 0,C 180,E1 26032.833,E2 26032.833} C_VEL
LIN {X 0,Y 570.832,Z 1126.128,A -85,B 0,C 180,E1 26030.71,E2 26030.71} C_VEL
LIN {X 0,Y 569.704,Z 1138.013,A -85,B 0,C 180,E1 26028.1,E2 26028.1} C_VEL
LIN {X 0,Y 568.886,Z 1148.287,A -85,B 0,C 180,E1 26025.392,E2 26025.392} C_VEL
LIN {X 0,Y 568.452,Z 1155.631,A -85,B 0,C 180,E1 26023.116,E2 26023.116} C_VEL
LIN {X 0,Y 568.157,Z 1161.717,A -85,B 0,C 180,E1 26020.855,E2 26020.855} C_VEL
LIN {X 0,Y 568.023,Z 1166.611,A -85,B 0,C 180,E1 26018.606,E2 26018.606} C_VEL
LIN {X 0,Y 567.949,Z 1170.356,A -85,B 0,C 180,E1 26016.369,E2 26016.369} C_VEL
LIN {X 0,Y 567.918,Z 1172.98,A -85,B 0,C 180,E1 26014.141,E2 26014.141} C_VEL
LIN {X 0,Y 567.909,Z 1174.547,A -85,B 0,C 180,E1 26011.817,E2 26011.817} C_VEL
LIN {X 0,Y 567.896,Z 1174.921,A -85,B 0,C 180,E1 26009.295,E2 26009.295} C_VEL
LIN {X 0,Y 567.913,Z 1173.641,A -85,B 0,C 180,E1 26006.468,E2 26006.468} C_VEL
LIN {X 0,Y 567.944,Z 1170.784,A -85,B 0,C 180,E1 26003.836,E2 26003.836} C_VEL
LIN {X 0,Y 568.014,Z 1166.987,A -85,B 0,C 180,E1 26001.498,E2 26001.498} C_VEL
LIN {X 0,Y 568.143,Z 1162.188,A -85,B 0,C 180,E1 25999.25,E2 25999.25} C_VEL
LIN {X 0,Y 568.422,Z 1156.2,A -85,B 0,C 180,E1 25996.989,E2 25996.989} C_VEL
LIN {X 0,Y 568.826,Z 1149.268,A -85,B 0,C 180,E1 25994.806,E2 25994.806} C_VEL
LIN {X 0,Y 569.41,Z 1141.247,A -85,B 0,C 180,E1 25992.633,E2 25992.633} C_VEL
LIN {X 0,Y 570.304,Z 1131.473,A -85,B 0,C 180,E1 25990.33,E2 25990.33} C_VEL
LIN {X 0,Y 571.803,Z 1117.406,A -85,B 0,C 180,E1 25987.485,E2 25987.485} C_VEL
LIN {X 0,Y 573.344,Z 1104.714,A -85,B 0,C 180,E1 25985.259,E2 25985.259} C_VEL
LIN {X 0,Y 575.099,Z 1091.823,A -85,B 0,C 180,E1 25983.238,E2 25983.238} C_VEL
LIN {X 0,Y 577.123,Z 1077.672,A -85,B 0,C 180,E1 25981.243,E2 25981.243} C_VEL
LIN {X 0,Y 579.947,Z 1059.604,A -85,B 0,C 180,E1 25978.969,E2 25978.969} C_VEL
LIN {X 0,Y 583.023,Z 1040.016,A -85,B 0,C 180,E1 25976.817,E2 25976.817} C_VEL
LIN {X 0,Y 585.885,Z 1022.16,A -85,B 0,C 180,E1 25975.072,E2 25975.072} C_VEL
LIN {X 0,Y 588.707,Z 1004.568,A -85,B 0,C 180,E1 25973.528,E2 25973.528} C_VEL
LIN {X 0,Y 591.594,Z 986.445,A -85,B 0,C 180,E1 25972.102,E2 25972.102} C_VEL
LIN {X 0,Y 594.626,Z 966.84,A -85,B 0,C 180,E1 25970.723,E2 25970.723} C_VEL
LIN {X 0,Y 597.72,Z 945.398,A -85,B 0,C 180,E1 25969.405,E2 25969.405} C_VEL
LIN {X 0,Y 600.615,Z 919.581,A -85,B 0,C 180,E1 25968.122,E2 25968.122} C_VEL
LIN {X 0,Y 602.889,Z 896.866,A -85,B 0,C 180,E1 25967.16,E2 25967.16} C_VEL
LIN {X 0,Y 604.758,Z 875.936,A -85,B 0,C 180,E1 25966.401,E2 25966.401} C_VEL
LIN {X 0,Y 606.334,Z 855.685,A -85,B 0,C 180,E1 25965.778,E2 25965.778} C_VEL
LIN {X 0,Y 608.106,Z 828.667,A -85,B 0,C 180,E1 25965.105,E2 25965.105} C_VEL
LIN {X 0,Y 609.269,Z 803.077,A -85,B 0,C 180,E1 25964.635,E2 25964.635} C_VEL
LIN {X 0,Y 614.305,Z 648.434,A -85,B 0,C 180,E1 25962.349,E2 25962.349} C_VEL
LIN {X 0,Y 622.672,Z 451.305,A -85,B 0,C 180,E1 25959.303,E2 25959.303} C_VEL
LIN {X 0,Y 624.282,Z 405.964,A -85,B 0,C 180,E1 25958.627,E2 25958.627} C_VEL
LIN {X 0,Y 613.583,Z 395.353,A -85,B 0,C 180,E1 25957.14,E2 25957.14} C_VEL
LIN {X 0,Y 605.193,Z 387.566,A -85,B 0,C 180,E1 25955.911,E2 25955.911} C_VEL
LIN {X 0,Y 598.954,Z 381.86,A -85,B 0,C 180,E1 25954.951,E2 25954.951} C_VEL
LIN {X 0,Y 596.637,Z 379.816,A -85,B 0,C 180,E1 25954.561,E2 25954.561} C_VEL
LIN {X 0,Y 594.856,Z 376.303,A -85,B 0,C 180,E1 25953.459,E2 25953.459} C_VEL
LIN {X 0,Y 592.264,Z 371.517,A -85,B 0,C 180,E1 25951.785,E2 25951.785} C_VEL
LIN {X 0,Y 589.982,Z 367.486,A -85,B 0,C 180,E1 25950.197,E2 25950.197} C_VEL
LIN {X 0,Y 588.973,Z 365.939,A -85,B 0,C 180,E1 25949.494,E2 25949.494} C_VEL
LIN {X 0,Y 586.898,Z 361.928,A -85,B 0,C 180,E1 25947.717,E2 25947.717} C_VEL
LIN {X 0,Y 583.951,Z 357.249,A -85,B 0,C 180,E1 25945.02,E2 25945.02} C_VEL
LIN {X 0,Y 583.409,Z 355.931,A -85,B 0,C 180,E1 25944.289,E2 25944.289} C_VEL
LIN {X 0,Y 580.603,Z 351.475,A -85,B 0,C 180,E1 25940.463,E2 25940.463} C_VEL
LIN {X 0,Y 580.173,Z 350.457,A -85,B 0,C 180,E1 25939.428,E2 25939.428} C_VEL
LIN {X 0,Y 578.652,Z 349.023,A -85,B 0,C 180,E1 25934.92,E2 25934.92} C_VEL
LIN {X 0,Y 579.156,Z 349.578,A -85,B 0,C 180,E1 25930.948,E2 25930.948} C_VEL
LIN {X 0,Y 580.51,Z 350.946,A -85,B 0,C 180,E1 25928.219,E2 25928.219} C_VEL
LIN {X 0,Y 583.519,Z 356.04,A -85,B 0,C 180,E1 25923.93,E2 25923.93} C_VEL
LIN {X 0,Y 586.349,Z 361.1,A -85,B 0,C 180,E1 25921.075,E2 25921.075} C_VEL
LIN {X 0,Y 587.085,Z 362.194,A -85,B 0,C 180,E1 25920.488,E2 25920.488} C_VEL
LIN {X 0,Y 589.235,Z 366.153,A -85,B 0,C 180,E1 25918.736,E2 25918.736} C_VEL
LIN {X 0,Y 590.127,Z 367.388,A -85,B 0,C 180,E1 25918.155,E2 25918.155} C_VEL
LIN {X 0,Y 592.505,Z 371.646,A -85,B 0,C 180,E1 25916.517,E2 25916.517} C_VEL
LIN {X 0,Y 596.055,Z 378.093,A -85,B 0,C 180,E1 25914.32,E2 25914.32} C_VEL
LIN {X 0,Y 598.91,Z 383.38,A -85,B 0,C 180,E1 25912.71,E2 25912.71} C_VEL
LIN {X 0,Y 601.626,Z 388.353,A -85,B 0,C 180,E1 25911.301,E2 25911.301} C_VEL
LIN {X 0,Y 606.084,Z 396.638,A -85,B 0,C 180,E1 25909.16,E2 25909.16} C_VEL
LIN {X 0,Y 612.509,Z 409.275,A -85,B 0,C 180,E1 25906.308,E2 25906.308} C_VEL
LIN {X 0,Y 618.909,Z 422.68,A -85,B 0,C 180,E1 25903.674,E2 25903.674} C_VEL
LIN {X 0,Y 621.468,Z 428.556,A -85,B 0,C 180,E1 25902.635,E2 25902.635} C_VEL
LIN {X 0,Y 617.127,Z 460.678,A -85,B 0,C 180,E1 25899.91,E2 25899.91} C_VEL
LIN {X 0,Y 612.638,Z 496.041,A -85,B 0,C 180,E1 25897.041,E2 25897.041} C_VEL
LIN {X 0,Y 608.202,Z 533.485,A -85,B 0,C 180,E1 25894.12,E2 25894.12} C_VEL
LIN {X 0,Y 602.986,Z 585.981,A -85,B 0,C 180,E1 25890.137,E2 25890.137} C_VEL
LIN {X 0,Y 603.319,Z 603.081,A -85,B 0,C 180,E1 25888.697,E2 25888.697} C_VEL
LIN {X 0,Y 605.537,Z 618.442,A -85,B 0,C 180,E1 25887.263,E2 25887.263} C_VEL
LIN {X 0,Y 609.793,Z 632.835,A -85,B 0,C 180,E1 25885.776,E2 25885.776} C_VEL
LIN {X 0,Y 615.802,Z 645.361,A -85,B 0,C 180,E1 25884.344,E2 25884.344} C_VEL
LIN {X 0,Y 623.135,Z 656.005,A -85,B 0,C 180,E1 25883.006,E2 25883.006} C_VEL
LIN {X 0,Y 632.768,Z 665.977,A -85,B 0,C 180,E1 25881.61,E2 25881.61} C_VEL
LIN {X 0,Y 643.636,Z 674.151,A -85,B 0,C 180,E1 25880.32,E2 25880.32} C_VEL
LIN {X 0,Y 655.592,Z 680.705,A -85,B 0,C 180,E1 25879.133,E2 25879.133} C_VEL
LIN {X 0,Y 663.856,Z 684.303,A -85,B 0,C 180,E1 25878.407,E2 25878.407} C_VEL
LIN {X 0,Y 649.784,Z 701.421,A -85,B 0,C 180,E1 25878.138,E2 25878.138} C_VEL
LIN {X 0,Y 641.343,Z 713.654,A -85,B 0,C 180,E1 25877.842,E2 25877.842} C_VEL
LIN {X 0,Y 638.446,Z 718.018,A -85,B 0,C 180,E1 25877.728,E2 25877.728} C_VEL
LIN {X 0,Y 629.684,Z 730.044,A -85,B 0,C 180,E1 25877.457,E2 25877.457} C_VEL
LIN {X 0,Y 622.605,Z 742.044,A -85,B 0,C 180,E1 25877.079,E2 25877.079} C_VEL
LIN {X 0,Y 616.063,Z 754.585,A -85,B 0,C 180,E1 25876.652,E2 25876.652} C_VEL
LIN {X 0,Y 614.32,Z 771.097,A -85,B 0,C 180,E1 25876.554,E2 25876.554} C_VEL
LIN {X 0,Y 612.786,Z 821.929,A -85,B 0,C 180,E1 25875.834,E2 25875.834} C_VEL
LIN {X 0,Y 610.888,Z 851.331,A -85,B 0,C 180,E1 25875.283,E2 25875.283} C_VEL
LIN {X 0,Y 608.728,Z 878.313,A -85,B 0,C 180,E1 25874.61,E2 25874.61} C_VEL
LIN {X 0,Y 606.332,Z 904.047,A -85,B 0,C 180,E1 25873.802,E2 25873.802} C_VEL
LIN {X 0,Y 603.642,Z 929.21,A -85,B 0,C 180,E1 25872.838,E2 25872.838} C_VEL
LIN {X 0,Y 600.466,Z 955.377,A -85,B 0,C 180,E1 25871.635,E2 25871.635} C_VEL
LIN {X 0,Y 597.241,Z 979.581,A -85,B 0,C 180,E1 25870.319,E2 25870.319} C_VEL
LIN {X 0,Y 593.913,Z 1001.837,A -85,B 0,C 180,E1 25868.898,E2 25868.898} C_VEL
LIN {X 0,Y 590.299,Z 1024.957,A -85,B 0,C 180,E1 25867.206,E2 25867.206} C_VEL
LIN {X 0,Y 586.812,Z 1046.523,A -85,B 0,C 180,E1 25865.402,E2 25865.402} C_VEL
LIN {X 0,Y 583.644,Z 1066.148,A -85,B 0,C 180,E1 25863.537,E2 25863.537} C_VEL
LIN {X 0,Y 580.423,Z 1086.422,A -85,B 0,C 180,E1 25861.347,E2 25861.347} C_VEL
LIN {X 0,Y 577.708,Z 1103.941,A -85,B 0,C 180,E1 25859.213,E2 25859.213} C_VEL
LIN {X 0,Y 575.248,Z 1120.847,A -85,B 0,C 180,E1 25856.866,E2 25856.866} C_VEL
LIN {X 0,Y 573.31,Z 1135.167,A -85,B 0,C 180,E1 25854.633,E2 25854.633} C_VEL
LIN {X 0,Y 571.578,Z 1149.443,A -85,B 0,C 180,E1 25852.091,E2 25852.091} C_VEL
LIN {X 0,Y 570.226,Z 1162.236,A -85,B 0,C 180,E1 25849.459,E2 25849.459} C_VEL
LIN {X 0,Y 569.295,Z 1172.786,A -85,B 0,C 180,E1 25846.95,E2 25846.95} C_VEL
LIN {X 0,Y 568.638,Z 1182.341,A -85,B 0,C 180,E1 25844.25,E2 25844.25} C_VEL
LIN {X 0,Y 568.25,Z 1189.804,A -85,B 0,C 180,E1 25841.673,E2 25841.673} C_VEL
LIN {X 0,Y 568.035,Z 1195.957,A -85,B 0,C 180,E1 25839.012,E2 25839.012} C_VEL
LIN {X 0,Y 567.949,Z 1200.352,A -85,B 0,C 180,E1 25836.468,E2 25836.468} C_VEL
LIN {X 0,Y 567.913,Z 1203.331,A -85,B 0,C 180,E1 25833.835,E2 25833.835} C_VEL
LIN {X 0,Y 567.917,Z 1204.783,A -85,B 0,C 180,E1 25831.209,E2 25831.209} C_VEL
LIN {X 0,Y 567.914,Z 1204.805,A -85,B 0,C 180,E1 25828.889,E2 25828.889} C_VEL
LIN {X 0,Y 567.912,Z 1203.417,A -85,B 0,C 180,E1 25826.264,E2 25826.264} C_VEL
LIN {X 0,Y 567.945,Z 1200.644,A -85,B 0,C 180,E1 25823.732,E2 25823.732} C_VEL
LIN {X 0,Y 568.029,Z 1196.148,A -85,B 0,C 180,E1 25821.088,E2 25821.088} C_VEL
LIN {X 0,Y 568.236,Z 1190.067,A -85,B 0,C 180,E1 25818.427,E2 25818.427} C_VEL
LIN {X 0,Y 568.622,Z 1182.679,A -85,B 0,C 180,E1 25815.851,E2 25815.851} C_VEL
LIN {X 0,Y 569.266,Z 1173.186,A -85,B 0,C 180,E1 25813.152,E2 25813.152} C_VEL
LIN {X 0,Y 570.183,Z 1162.684,A -85,B 0,C 180,E1 25810.641,E2 25810.641} C_VEL
LIN {X 0,Y 571.52,Z 1149.984,A -85,B 0,C 180,E1 25808.011,E2 25808.011} C_VEL
LIN {X 0,Y 573.229,Z 1135.797,A -85,B 0,C 180,E1 25805.471,E2 25805.471} C_VEL
LIN {X 0,Y 575.151,Z 1121.547,A -85,B 0,C 180,E1 25803.238,E2 25803.238} C_VEL
LIN {X 0,Y 577.586,Z 1104.767,A -85,B 0,C 180,E1 25800.891,E2 25800.891} C_VEL
LIN {X 0,Y 580.339,Z 1086.946,A -85,B 0,C 180,E1 25798.714,E2 25798.714} C_VEL
LIN {X 0,Y 583.488,Z 1067.208,A -85,B 0,C 180,E1 25796.569,E2 25796.569} C_VEL
LIN {X 0,Y 586.716,Z 1047.078,A -85,B 0,C 180,E1 25794.648,E2 25794.648} C_VEL
LIN {X 0,Y 590.196,Z 1025.602,A -85,B 0,C 180,E1 25792.844,E2 25792.844} C_VEL
LIN {X 0,Y 593.691,Z 1003.371,A -85,B 0,C 180,E1 25791.205,E2 25791.205} C_VEL
LIN {X 0,Y 596.961,Z 981.526,A -85,B 0,C 180,E1 25789.799,E2 25789.799} C_VEL
LIN {X 0,Y 600.217,Z 957.406,A -85,B 0,C 180,E1 25788.469,E2 25788.469} C_VEL
LIN {X 0,Y 603.377,Z 931.475,A -85,B 0,C 180,E1 25787.258,E2 25787.258} C_VEL
LIN {X 0,Y 606.248,Z 904.864,A -85,B 0,C 180,E1 25786.226,E2 25786.226} C_VEL
LIN {X 0,Y 608.845,Z 877.375,A -85,B 0,C 180,E1 25785.36,E2 25785.36} C_VEL
LIN {X 0,Y 611.083,Z 849.119,A -85,B 0,C 180,E1 25784.666,E2 25784.666} C_VEL
LIN {X 0,Y 612.977,Z 818.419,A -85,B 0,C 180,E1 25784.109,E2 25784.109} C_VEL
LIN {X 0,Y 615.35,Z 742.983,A -85,B 0,C 180,E1 25783.051,E2 25783.051} C_VEL
LIN {X 0,Y 622.427,Z 660.589,A -85,B 0,C 180,E1 25781.664,E2 25781.664} C_VEL
LIN {X 0,Y 623.842,Z 645.075,A -85,B 0,C 180,E1 25781.41,E2 25781.41} C_VEL
LIN {X 0,Y 627.058,Z 610.933,A -85,B 0,C 180,E1 25780.862,E2 25780.862} C_VEL
LIN {X 0,Y 628.757,Z 595.046,A -85,B 0,C 180,E1 25780.627,E2 25780.627} C_VEL
LIN {X 0,Y 631.193,Z 566.944,A -85,B 0,C 180,E1 25780.155,E2 25780.155} C_VEL
LIN {X 0,Y 634.701,Z 537.252,A -85,B 0,C 180,E1 25779.75,E2 25779.75} C_VEL
LIN {X 0,Y 636.694,Z 512.777,A -85,B 0,C 180,E1 25779.326,E2 25779.326} C_VEL
LIN {X 0,Y 641.004,Z 479.003,A -85,B 0,C 180,E1 25778.9,E2 25778.9} C_VEL
LIN {X 0,Y 641.535,Z 473.11,A -85,B 0,C 180,E1 25778.803,E2 25778.803} C_VEL
LIN {X 0,Y 643.257,Z 451.315,A -85,B 0,C 180,E1 25778.42,E2 25778.42} C_VEL
LIN {X 0,Y 645.134,Z 435.267,A -85,B 0,C 180,E1 25778.2,E2 25778.2} C_VEL
LIN {X 0,Y 635.546,Z 424.708,A -85,B 0,C 180,E1 25776.885,E2 25776.885} C_VEL
LIN {X 0,Y 617.937,Z 398.41,A -85,B 0,C 180,E1 25774.047,E2 25774.047} C_VEL
LIN {X 0,Y 606.98,Z 382.962,A -85,B 0,C 180,E1 25772.119,E2 25772.119} C_VEL
LIN {X 0,Y 598.722,Z 371.795,A -85,B 0,C 180,E1 25770.566,E2 25770.566} C_VEL
LIN {X 0,Y 595.319,Z 367.243,A -85,B 0,C 180,E1 25769.896,E2 25769.896} C_VEL
LIN {X 0,Y 591.659,Z 362.389,A -85,B 0,C 180,E1 25769.153,E2 25769.153} C_VEL
LIN {X 0,Y 587.432,Z 356.983,A -85,B 0,C 180,E1 25768.27,E2 25768.27} C_VEL
LIN {X 0,Y 584.15,Z 352.672,A -85,B 0,C 180,E1 25767.554,E2 25767.554} C_VEL
LIN {X 0,Y 582.81,Z 351.119,A -85,B 0,C 180,E1 25767.263,E2 25767.263} C_VEL
LIN {X 0,Y 579.799,Z 347.386,A -85,B 0,C 180,E1 25766.585,E2 25766.585} C_VEL
LIN {X 0,Y 578.671,Z 345.584,A -85,B 0,C 180,E1 25766.309,E2 25766.309} C_VEL
LIN {X 0,Y 575.555,Z 342.466,A -85,B 0,C 180,E1 25765.604,E2 25765.604} C_VEL
LIN {X 0,Y 574.086,Z 339.573,A -85,B 0,C 180,E1 25765.204,E2 25765.204} C_VEL
LIN {X 0,Y 571.082,Z 337.262,A -85,B 0,C 180,E1 25764.517,E2 25764.517} C_VEL
LIN {X 0,Y 569.564,Z 334.233,A -85,B 0,C 180,E1 25764.08,E2 25764.08} C_VEL
LIN {X 0,Y 569.375,Z 333.244,A -85,B 0,C 180,E1 25763.966,E2 25763.966} C_VEL
LIN {X 0,Y 569.376,Z 333.287,A -85,B 0,C 180,E1 25760.67,E2 25760.67} C_VEL
LIN {X 0,Y 569.374,Z 333.286,A -85,B 0,C 180,E1 25757.159,E2 25757.159} C_VEL
LIN {X 0,Y 569.35,Z 333.316,A -85,B 0,C 180,E1 25754.983,E2 25754.983} C_VEL
LIN {X 0,Y 575.406,Z 351.887,A -85,B 0,C 180,E1 25754.098,E2 25754.098} C_VEL
LIN {X 0,Y 575.217,Z 433.702,A -85,B 0,C 180,E1 25751.201,E2 25751.201} C_VEL
LIN {X 0,Y 575.469,Z 516.51,A -85,B 0,C 180,E1 25748.116,E2 25748.116} C_VEL
LIN {X 0,Y 575.274,Z 593.907,A -85,B 0,C 180,E1 25745.141,E2 25745.141} C_VEL
LIN {X 0,Y 574.663,Z 670.916,A -85,B 0,C 180,E1 25742.094,E2 25742.094} C_VEL
LIN {X 0,Y 573.819,Z 745.321,A -85,B 0,C 180,E1 25739.101,E2 25739.101} C_VEL
LIN {X 0,Y 572.798,Z 824.725,A -85,B 0,C 180,E1 25735.846,E2 25735.846} C_VEL
LIN {X 0,Y 572.182,Z 850.563,A -85,B 0,C 180,E1 25734.786,E2 25734.786} C_VEL
LIN {X 0,Y 571.705,Z 857.724,A -85,B 0,C 180,E1 25734.526,E2 25734.526} C_VEL
LIN {X 0,Y 571.006,Z 971.664,A -85,B 0,C 180,E1 25732.994,E2 25732.994} C_VEL
LIN {X 0,Y 571.037,Z 984.062,A -85,B 0,C 180,E1 25732.697,E2 25732.697} C_VEL
LIN {X 0,Y 571.002,Z 995.515,A -85,B 0,C 180,E1 25732.301,E2 25732.301} C_VEL
LIN {X 0,Y 570.876,Z 1008.658,A -85,B 0,C 180,E1 25731.692,E2 25731.692} C_VEL
LIN {X 0,Y 570.634,Z 1021.506,A -85,B 0,C 180,E1 25730.876,E2 25730.876} C_VEL
LIN {X 0,Y 570.414,Z 1031.094,A -85,B 0,C 180,E1 25730.108,E2 25730.108} C_VEL
LIN {X 0,Y 570.177,Z 1039.514,A -85,B 0,C 180,E1 25729.287,E2 25729.287} C_VEL
LIN {X 0,Y 569.936,Z 1047.318,A -85,B 0,C 180,E1 25728.36,E2 25728.36} C_VEL
LIN {X 0,Y 569.671,Z 1055.666,A -85,B 0,C 180,E1 25727.12,E2 25727.12} C_VEL
LIN {X 0,Y 569.44,Z 1061.857,A -85,B 0,C 180,E1 25725.873,E2 25725.873} C_VEL
LIN {X 0,Y 569.294,Z 1066.132,A -85,B 0,C 180,E1 25724.725,E2 25724.725} C_VEL
LIN {X 0,Y 569.183,Z 1069.168,A -85,B 0,C 180,E1 25723.571,E2 25723.571} C_VEL
LIN {X 0,Y 569.117,Z 1071.032,A -85,B 0,C 180,E1 25722.411,E2 25722.411} C_VEL
LIN {X 0,Y 569.075,Z 1071.837,A -85,B 0,C 180,E1 25720.961,E2 25720.961} C_VEL
LIN {X 0,Y 569.077,Z 1070.686,A -85,B 0,C 180,E1 25719.473,E2 25719.473} C_VEL
LIN {X 0,Y 569.112,Z 1068.377,A -85,B 0,C 180,E1 25718.24,E2 25718.24} C_VEL
LIN {X 0,Y 569.198,Z 1064.889,A -85,B 0,C 180,E1 25717.047,E2 25717.047} C_VEL
LIN {X 0,Y 569.363,Z 1059.41,A -85,B 0,C 180,E1 25715.707,E2 25715.707} C_VEL
LIN {X 0,Y 569.582,Z 1052.096,A -85,B 0,C 180,E1 25714.415,E2 25714.415} C_VEL
LIN {X 0,Y 569.817,Z 1044.534,A -85,B 0,C 180,E1 25713.362,E2 25713.362} C_VEL
LIN {X 0,Y 570.069,Z 1036.182,A -85,B 0,C 180,E1 25712.416,E2 25712.416} C_VEL
LIN {X 0,Y 570.392,Z 1025.218,A -85,B 0,C 180,E1 25711.408,E2 25711.408} C_VEL
LIN {X 0,Y 570.643,Z 1013.214,A -85,B 0,C 180,E1 25710.559,E2 25710.559} C_VEL
LIN {X 0,Y 570.85,Z 1002.129,A -85,B 0,C 180,E1 25709.937,E2 25709.937} C_VEL
LIN {X 0,Y 571.001,Z 990.37,A -85,B 0,C 180,E1 25709.423,E2 25709.423} C_VEL
LIN {X 0,Y 571.098,Z 975.934,A -85,B 0,C 180,E1 25708.964,E2 25708.964} C_VEL
LIN {X 0,Y 571.062,Z 959.003,A -85,B 0,C 180,E1 25708.66,E2 25708.66} C_VEL
LIN {X 0,Y 571.9,Z 851.664,A -85,B 0,C 180,E1 25707.243,E2 25707.243} C_VEL
LIN {X 0,Y 572.541,Z 834.115,A -85,B 0,C 180,E1 25706.505,E2 25706.505} C_VEL
LIN {X 0,Y 573.35,Z 786.217,A -85,B 0,C 180,E1 25704.461,E2 25704.461} C_VEL
LIN {X 0,Y 572.552,Z 779.218,A -85,B 0,C 180,E1 25704.133,E2 25704.133} C_VEL
LIN {X 0,Y 566.686,Z 760.145,A -85,B 0,C 180,E1 25703.117,E2 25703.117} C_VEL
LIN {X 0,Y 566.241,Z 755.107,A -85,B 0,C 180,E1 25702.885,E2 25702.885} C_VEL
LIN {X 0,Y 567.138,Z 711.494,A -85,B 0,C 180,E1 25700.993,E2 25700.993} C_VEL
LIN {X 0,Y 568.218,Z 712.944,A -85,B 0,C 180,E1 25700.822,E2 25700.822} C_VEL
LIN {X 0,Y 570.036,Z 712.678,A -85,B 0,C 180,E1 25700.614,E2 25700.614} C_VEL
LIN {X 0,Y 572.948,Z 709.852,A -85,B 0,C 180,E1 25700.351,E2 25700.351} C_VEL
LIN {X 0,Y 576.632,Z 703.829,A -85,B 0,C 180,E1 25700.09,E2 25700.09} C_VEL
LIN {X 0,Y 580.15,Z 702.228,A -85,B 0,C 180,E1 25699.735,E2 25699.735} C_VEL
LIN {X 0,Y 583.993,Z 698.391,A -85,B 0,C 180,E1 25699.411,E2 25699.411} C_VEL
LIN {X 0,Y 587.296,Z 693.684,A -85,B 0,C 180,E1 25699.173,E2 25699.173} C_VEL
LIN {X 0,Y 591.766,Z 690.653,A -85,B 0,C 180,E1 25698.778,E2 25698.778} C_VEL
LIN {X 0,Y 596.485,Z 685.356,A -85,B 0,C 180,E1 25698.424,E2 25698.424} C_VEL
LIN {X 0,Y 598.238,Z 683.227,A -85,B 0,C 180,E1 25698.301,E2 25698.301} C_VEL
LIN {X 0,Y 603.568,Z 679.216,A -85,B 0,C 180,E1 25697.892,E2 25697.892} C_VEL
LIN {X 0,Y 607.316,Z 675.461,A -85,B 0,C 180,E1 25697.652,E2 25697.652} C_VEL
LIN {X 0,Y 603.387,Z 784.358,A -85,B 0,C 180,E1 25695.991,E2 25695.991} C_VEL
LIN {X 0,Y 601.912,Z 818.698,A -85,B 0,C 180,E1 25695.425,E2 25695.425} C_VEL
LIN {X 0,Y 600.352,Z 844.558,A -85,B 0,C 180,E1 25694.84,E2 25694.84} C_VEL
LIN {X 0,Y 598.303,Z 872.094,A -85,B 0,C 180,E1 25694.046,E2 25694.046} C_VEL
LIN {X 0,Y 596.216,Z 895.747,A -85,B 0,C 180,E1 25693.21,E2 25693.21} C_VEL
LIN {X 0,Y 594.474,Z 913.375,A -85,B 0,C 180,E1 25692.479,E2 25692.479} C_VEL
LIN {X 0,Y 592.178,Z 933.884,A -85,B 0,C 180,E1 25691.51,E2 25691.51} C_VEL
LIN {X 0,Y 589.371,Z 956.655,A -85,B 0,C 180,E1 25690.27,E2 25690.27} C_VEL
LIN {X 0,Y 586.358,Z 978.898,A -85,B 0,C 180,E1 25688.869,E2 25688.869} C_VEL
LIN {X 0,Y 582.511,Z 1001.677,A -85,B 0,C 180,E1 25687.111,E2 25687.111} C_VEL
LIN {X 0,Y 579.472,Z 1019.521,A -85,B 0,C 180,E1 25685.557,E2 25685.557} C_VEL
LIN {X 0,Y 576.538,Z 1036.759,A -85,B 0,C 180,E1 25683.883,E2 25683.883} C_VEL
LIN {X 0,Y 573.771,Z 1053.192,A -85,B 0,C 180,E1 25682.109,E2 25682.109} C_VEL
LIN {X 0,Y 570.872,Z 1071.112,A -85,B 0,C 180,E1 25679.947,E2 25679.947} C_VEL
LIN {X 0,Y 568.001,Z 1089.076,A -85,B 0,C 180,E1 25677.466,E2 25677.466} C_VEL
LIN {X 0,Y 566.109,Z 1102.225,A -85,B 0,C 180,E1 25675.418,E2 25675.418} C_VEL
LIN {X 0,Y 564.514,Z 1113.995,A -85,B 0,C 180,E1 25673.377,E2 25673.377} C_VEL
LIN {X 0,Y 563.242,Z 1124.505,A -85,B 0,C 180,E1 25671.342,E2 25671.342} C_VEL
LIN {X 0,Y 562.225,Z 1133.853,A -85,B 0,C 180,E1 25669.318,E2 25669.318} C_VEL
LIN {X 0,Y 561.412,Z 1142.519,A -85,B 0,C 180,E1 25667.198,E2 25667.198} C_VEL
LIN {X 0,Y 560.828,Z 1150.407,A -85,B 0,C 180,E1 25664.983,E2 25664.983} C_VEL
LIN {X 0,Y 560.351,Z 1158.03,A -85,B 0,C 180,E1 25662.47,E2 25662.47} C_VEL
LIN {X 0,Y 560.078,Z 1165.035,A -85,B 0,C 180,E1 25659.558,E2 25659.558} C_VEL
LIN {X 0,Y 559.958,Z 1169.62,A -85,B 0,C 180,E1 25656.975,E2 25656.975} C_VEL
LIN {X 0,Y 559.917,Z 1172.588,A -85,B 0,C 180,E1 25654.61,E2 25654.61} C_VEL
LIN {X 0,Y 559.908,Z 1174.301,A -85,B 0,C 180,E1 25652.355,E2 25652.355} C_VEL
LIN {X 0,Y 559.915,Z 1174.918,A -85,B 0,C 180,E1 25650.001,E2 25650.001} C_VEL
LIN {X 0,Y 559.908,Z 1174.296,A -85,B 0,C 180,E1 25647.545,E2 25647.545} C_VEL
LIN {X 0,Y 559.918,Z 1172.479,A -85,B 0,C 180,E1 25645.184,E2 25645.184} C_VEL
LIN {X 0,Y 559.973,Z 1169.162,A -85,B 0,C 180,E1 25642.615,E2 25642.615} C_VEL
LIN {X 0,Y 560.124,Z 1163.665,A -85,B 0,C 180,E1 25639.718,E2 25639.718} C_VEL
LIN {X 0,Y 560.413,Z 1157.095,A -85,B 0,C 180,E1 25637.115,E2 25637.115} C_VEL
LIN {X 0,Y 560.85,Z 1150.01,A -85,B 0,C 180,E1 25634.808,E2 25634.808} C_VEL
LIN {X 0,Y 561.459,Z 1142.058,A -85,B 0,C 180,E1 25632.593,E2 25632.593} C_VEL
LIN {X 0,Y 562.284,Z 1133.324,A -85,B 0,C 180,E1 25630.471,E2 25630.471} C_VEL
LIN {X 0,Y 563.314,Z 1123.901,A -85,B 0,C 180,E1 25628.445,E2 25628.445} C_VEL
LIN {X 0,Y 564.6,Z 1113.317,A -85,B 0,C 180,E1 25626.409,E2 25626.409} C_VEL
LIN {X 0,Y 566.387,Z 1100.166,A -85,B 0,C 180,E1 25624.15,E2 25624.15} C_VEL
LIN {X 0,Y 569.095,Z 1082.175,A -85,B 0,C 180,E1 25621.454,E2 25621.454} C_VEL
LIN {X 0,Y 571.542,Z 1066.586,A -85,B 0,C 180,E1 25619.399,E2 25619.399} C_VEL
LIN {X 0,Y 573.972,Z 1051.952,A -85,B 0,C 180,E1 25617.661,E2 25617.661} C_VEL
LIN {X 0,Y 576.74,Z 1035.596,A -85,B 0,C 180,E1 25615.908,E2 25615.908} C_VEL
LIN {X 0,Y 579.729,Z 1018.09,A -85,B 0,C 180,E1 25614.221,E2 25614.221} C_VEL
LIN {X 0,Y 583.621,Z 995.515,A -85,B 0,C 180,E1 25612.295,E2 25612.295} C_VEL
LIN {X 0,Y 586.871,Z 975.26,A -85,B 0,C 180,E1 25610.797,E2 25610.797} C_VEL
LIN {X 0,Y 589.567,Z 955.096,A -85,B 0,C 180,E1 25609.551,E2 25609.551} C_VEL
LIN {X 0,Y 592.247,Z 933.279,A -85,B 0,C 180,E1 25608.37,E2 25608.37} C_VEL
LIN {X 0,Y 594.615,Z 912.119,A -85,B 0,C 180,E1 25607.376,E2 25607.376} C_VEL
LIN {X 0,Y 596.32,Z 894.538,A -85,B 0,C 180,E1 25606.656,E2 25606.656} C_VEL
LIN {X 0,Y 598.234,Z 872.584,A -85,B 0,C 180,E1 25605.884,E2 25605.884} C_VEL
LIN {X 0,Y 600.321,Z 844.579,A -85,B 0,C 180,E1 25605.075,E2 25605.075} C_VEL
LIN {X 0,Y 601.66,Z 822.595,A -85,B 0,C 180,E1 25604.57,E2 25604.57} C_VEL
LIN {X 0,Y 602.726,Z 801.138,A -85,B 0,C 180,E1 25604.177,E2 25604.177} C_VEL
LIN {X 0,Y 607.111,Z 678.905,A -85,B 0,C 180,E1 25602.318,E2 25602.318} C_VEL
LIN {X 0,Y 616.307,Z 483.491,A -85,B 0,C 180,E1 25599.212,E2 25599.212} C_VEL
LIN {X 0,Y 619.044,Z 410.604,A -85,B 0,C 180,E1 25598.099,E2 25598.099} C_VEL
LIN {X 0,Y 609.681,Z 401.536,A -85,B 0,C 180,E1 25596.771,E2 25596.771} C_VEL
LIN {X 0,Y 602.436,Z 394.713,A -85,B 0,C 180,E1 25595.69,E2 25595.69} C_VEL
LIN {X 0,Y 596.149,Z 388.959,A -85,B 0,C 180,E1 25594.71,E2 25594.71} C_VEL
LIN {X 0,Y 591.043,Z 384.223,A -85,B 0,C 180,E1 25593.839,E2 25593.839} C_VEL
LIN {X 0,Y 587.573,Z 377.88,A -85,B 0,C 180,E1 25591.61,E2 25591.61} C_VEL
LIN {X 0,Y 585.393,Z 373.762,A -85,B 0,C 180,E1 25590.008,E2 25590.008} C_VEL
LIN {X 0,Y 582.533,Z 368.791,A -85,B 0,C 180,E1 25587.721,E2 25587.721} C_VEL
LIN {X 0,Y 581.493,Z 367.352,A -85,B 0,C 180,E1 25586.887,E2 25586.887} C_VEL
LIN {X 0,Y 579.463,Z 363.358,A -85,B 0,C 180,E1 25584.682,E2 25584.682} C_VEL
LIN {X 0,Y 578.546,Z 362.171,A -85,B 0,C 180,E1 25583.747,E2 25583.747} C_VEL
LIN {X 0,Y 575.989,Z 357.279,A -85,B 0,C 180,E1 25579.469,E2 25579.469} C_VEL
LIN {X 0,Y 574.461,Z 355.839,A -85,B 0,C 180,E1 25574.928,E2 25574.928} C_VEL
LIN {X 0,Y 574.972,Z 356.4,A -85,B 0,C 180,E1 25570.927,E2 25570.927} C_VEL
LIN {X 0,Y 576.299,Z 357.839,A -85,B 0,C 180,E1 25568.179,E2 25568.179} C_VEL
LIN {X 0,Y 579.581,Z 363.46,A -85,B 0,C 180,E1 25563.561,E2 25563.561} C_VEL
LIN {X 0,Y 581.79,Z 367.584,A -85,B 0,C 180,E1 25561.28,E2 25561.28} C_VEL
LIN {X 0,Y 582.672,Z 368.795,A -85,B 0,C 180,E1 25560.59,E2 25560.59} C_VEL
LIN {X 0,Y 584.792,Z 372.759,A -85,B 0,C 180,E1 25558.824,E2 25558.824} C_VEL
LIN {X 0,Y 585.764,Z 374.304,A -85,B 0,C 180,E1 25558.141,E2 25558.141} C_VEL
LIN {X 0,Y 588.594,Z 379.351,A -85,B 0,C 180,E1 25556.201,E2 25556.201} C_VEL
LIN {X 0,Y 591.525,Z 384.75,A -85,B 0,C 180,E1 25554.374,E2 25554.374} C_VEL
LIN {X 0,Y 594.206,Z 389.694,A -85,B 0,C 180,E1 25552.847,E2 25552.847} C_VEL
LIN {X 0,Y 597.056,Z 395.041,A -85,B 0,C 180,E1 25551.331,E2 25551.331} C_VEL
LIN {X 0,Y 601.287,Z 402.978,A -85,B 0,C 180,E1 25549.266,E2 25549.266} C_VEL
LIN {X 0,Y 607.645,Z 415.646,A -85,B 0,C 180,E1 25546.39,E2 25546.39} C_VEL
LIN {X 0,Y 613.767,Z 428.594,A -85,B 0,C 180,E1 25543.825,E2 25543.825} C_VEL
LIN {X 0,Y 615.898,Z 433.202,A -85,B 0,C 180,E1 25542.977,E2 25542.977} C_VEL
LIN {X 0,Y 611.396,Z 464.993,A -85,B 0,C 180,E1 25540.262,E2 25540.262} C_VEL
LIN {X 0,Y 606.762,Z 499.76,A -85,B 0,C 180,E1 25537.42,E2 25537.42} C_VEL
LIN {X 0,Y 602.103,Z 537.245,A -85,B 0,C 180,E1 25534.472,E2 25534.472} C_VEL
LIN {X 0,Y 596.675,Z 589.326,A -85,B 0,C 180,E1 25530.483,E2 25530.483} C_VEL
LIN {X 0,Y 596.946,Z 606.746,A -85,B 0,C 180,E1 25528.998,E2 25528.998} C_VEL
LIN {X 0,Y 599.075,Z 622.127,A -85,B 0,C 180,E1 25527.547,E2 25527.547} C_VEL
LIN {X 0,Y 603.207,Z 636.613,A -85,B 0,C 180,E1 25526.039,E2 25526.039} C_VEL
LIN {X 0,Y 609.067,Z 649.297,A -85,B 0,C 180,E1 25524.584,E2 25524.584} C_VEL
LIN {X 0,Y 616.729,Z 660.762,A -85,B 0,C 180,E1 25523.139,E2 25523.139} C_VEL
LIN {X 0,Y 626.259,Z 670.875,A -85,B 0,C 180,E1 25521.721,E2 25521.721} C_VEL
LIN {X 0,Y 637.005,Z 679.248,A -85,B 0,C 180,E1 25520.41,E2 25520.41} C_VEL
LIN {X 0,Y 649.511,Z 686.382,A -85,B 0,C 180,E1 25519.136,E2 25519.136} C_VEL
LIN {X 0,Y 653.128,Z 688.156,A -85,B 0,C 180,E1 25518.799,E2 25518.799} C_VEL
LIN {X 0,Y 641.714,Z 702.669,A -85,B 0,C 180,E1 25518.542,E2 25518.542} C_VEL
LIN {X 0,Y 632.929,Z 715.726,A -85,B 0,C 180,E1 25518.213,E2 25518.213} C_VEL
LIN {X 0,Y 623.682,Z 728.493,A -85,B 0,C 180,E1 25517.924,E2 25517.924} C_VEL
LIN {X 0,Y 616.587,Z 740.502,A -85,B 0,C 180,E1 25517.546,E2 25517.546} C_VEL
LIN {X 0,Y 611.133,Z 750.853,A -85,B 0,C 180,E1 25517.203,E2 25517.203} C_VEL
LIN {X 0,Y 608.882,Z 769.888,A -85,B 0,C 180,E1 25517.114,E2 25517.114} C_VEL
LIN {X 0,Y 607.26,Z 819.917,A -85,B 0,C 180,E1 25516.404,E2 25516.404} C_VEL
LIN {X 0,Y 605.243,Z 850.062,A -85,B 0,C 180,E1 25515.842,E2 25515.842} C_VEL
LIN {X 0,Y 602.887,Z 878.139,A -85,B 0,C 180,E1 25515.14,E2 25515.14} C_VEL
LIN {X 0,Y 600.253,Z 904.721,A -85,B 0,C 180,E1 25514.294,E2 25514.294} C_VEL
LIN {X 0,Y 597.616,Z 928.65,A -85,B 0,C 180,E1 25513.376,E2 25513.376} C_VEL
LIN {X 0,Y 594.433,Z 953.914,A -85,B 0,C 180,E1 25512.219,E2 25512.219} C_VEL
LIN {X 0,Y 590.96,Z 978.971,A -85,B 0,C 180,E1 25510.859,E2 25510.859} C_VEL
LIN {X 0,Y 587.578,Z 1000.955,A -85,B 0,C 180,E1 25509.462,E2 25509.462} C_VEL
LIN {X 0,Y 583.913,Z 1023.601,A -85,B 0,C 180,E1 25507.807,E2 25507.807} C_VEL
LIN {X 0,Y 580.35,Z 1044.766,A -85,B 0,C 180,E1 25506.04,E2 25506.04} C_VEL
LIN {X 0,Y 576.94,Z 1064.528,A -85,B 0,C 180,E1 25504.159,E2 25504.159} C_VEL
LIN {X 0,Y 573.505,Z 1084.914,A -85,B 0,C 180,E1 25501.962,E2 25501.962} C_VEL
LIN {X 0,Y 570.808,Z 1101.4,A -85,B 0,C 180,E1 25499.948,E2 25499.948} C_VEL
LIN {X 0,Y 567.962,Z 1119.415,A -85,B 0,C 180,E1 25497.465,E2 25497.465} C_VEL
LIN {X 0,Y 565.89,Z 1133.86,A -85,B 0,C 180,E1 25495.201,E2 25495.201} C_VEL
LIN {X 0,Y 563.99,Z 1148.323,A -85,B 0,C 180,E1 25492.624,E2 25492.624} C_VEL
LIN {X 0,Y 562.509,Z 1161.296,A -85,B 0,C 180,E1 25489.954,E2 25489.954} C_VEL
LIN {X 0,Y 561.478,Z 1171.969,A -85,B 0,C 180,E1 25487.407,E2 25487.407} C_VEL
LIN {X 0,Y 560.77,Z 1181.3,A -85,B 0,C 180,E1 25484.771,E2 25484.771} C_VEL
LIN {X 0,Y 560.296,Z 1189.263,A -85,B 0,C 180,E1 25482.05,E2 25482.05} C_VEL
LIN {X 0,Y 560.059,Z 1195.564,A -85,B 0,C 180,E1 25479.349,E2 25479.349} C_VEL
LIN {X 0,Y 559.952,Z 1200.044,A -85,B 0,C 180,E1 25476.767,E2 25476.767} C_VEL
LIN {X 0,Y 559.917,Z 1203.153,A -85,B 0,C 180,E1 25474.095,E2 25474.095} C_VEL
LIN {X 0,Y 559.909,Z 1204.717,A -85,B 0,C 180,E1 25471.534,E2 25471.534} C_VEL
LIN {X 0,Y 559.906,Z 1204.845,A -85,B 0,C 180,E1 25469.078,E2 25469.078} C_VEL
LIN {X 0,Y 559.913,Z 1203.592,A -85,B 0,C 180,E1 25466.415,E2 25466.415} C_VEL
LIN {X 0,Y 559.941,Z 1200.908,A -85,B 0,C 180,E1 25463.848,E2 25463.848} C_VEL
LIN {X 0,Y 560.026,Z 1196.734,A -85,B 0,C 180,E1 25461.27,E2 25461.27} C_VEL
LIN {X 0,Y 560.21,Z 1191.143,A -85,B 0,C 180,E1 25458.676,E2 25458.676} C_VEL
LIN {X 0,Y 560.62,Z 1183.643,A -85,B 0,C 180,E1 25455.961,E2 25455.961} C_VEL
LIN {X 0,Y 561.308,Z 1173.961,A -85,B 0,C 180,E1 25453.119,E2 25453.119} C_VEL
LIN {X 0,Y 562.315,Z 1163.144,A -85,B 0,C 180,E1 25450.464,E2 25450.464} C_VEL
LIN {X 0,Y 563.663,Z 1151.104,A -85,B 0,C 180,E1 25447.909,E2 25447.909} C_VEL
LIN {X 0,Y 565.538,Z 1136.445,A -85,B 0,C 180,E1 25445.226,E2 25445.226} C_VEL
LIN {X 0,Y 567.658,Z 1121.547,A -85,B 0,C 180,E1 25442.856,E2 25442.856} C_VEL
LIN {X 0,Y 570.27,Z 1104.766,A -85,B 0,C 180,E1 25440.481,E2 25440.481} C_VEL
LIN {X 0,Y 573.164,Z 1086.981,A -85,B 0,C 180,E1 25438.282,E2 25438.282} C_VEL
LIN {X 0,Y 576.46,Z 1067.441,A -85,B 0,C 180,E1 25436.133,E2 25436.133} C_VEL
LIN {X 0,Y 579.818,Z 1047.658,A -85,B 0,C 180,E1 25434.224,E2 25434.224} C_VEL
LIN {X 0,Y 583.468,Z 1026.276,A -85,B 0,C 180,E1 25432.404,E2 25432.404} C_VEL
LIN {X 0,Y 587.007,Z 1004.91,A -85,B 0,C 180,E1 25430.805,E2 25430.805} C_VEL
LIN {X 0,Y 590.469,Z 982.343,A -85,B 0,C 180,E1 25429.344,E2 25429.344} C_VEL
LIN {X 0,Y 593.893,Z 958.038,A -85,B 0,C 180,E1 25427.991,E2 25427.991} C_VEL
LIN {X 0,Y 597.184,Z 932.366,A -85,B 0,C 180,E1 25426.779,E2 25426.779} C_VEL
LIN {X 0,Y 600.211,Z 905.67,A -85,B 0,C 180,E1 25425.732,E2 25425.732} C_VEL
LIN {X 0,Y 602.946,Z 877.94,A -85,B 0,C 180,E1 25424.85,E2 25424.85} C_VEL
LIN {X 0,Y 605.315,Z 849.333,A -85,B 0,C 180,E1 25424.141,E2 25424.141} C_VEL
LIN {X 0,Y 607.352,Z 818.474,A -85,B 0,C 180,E1 25423.572,E2 25423.572} C_VEL
LIN {X 0,Y 609.498,Z 748.207,A -85,B 0,C 180,E1 25422.588,E2 25422.588} C_VEL
LIN {X 0,Y 610.922,Z 727.519,A -85,B 0,C 180,E1 25422.246,E2 25422.246} C_VEL
LIN {X 0,Y 617.102,Z 658.887,A -85,B 0,C 180,E1 25421.101,E2 25421.101} C_VEL
LIN {X 0,Y 618.49,Z 643.085,A -85,B 0,C 180,E1 25420.834,E2 25420.834} C_VEL
LIN {X 0,Y 621.99,Z 607.885,A -85,B 0,C 180,E1 25420.28,E2 25420.28} C_VEL
LIN {X 0,Y 623.306,Z 595.328,A -85,B 0,C 180,E1 25420.089,E2 25420.089} C_VEL
LIN {X 0,Y 625.865,Z 566.693,A -85,B 0,C 180,E1 25419.609,E2 25419.609} C_VEL
LIN {X 0,Y 629.319,Z 537.782,A -85,B 0,C 180,E1 25419.214,E2 25419.214} C_VEL
LIN {X 0,Y 631.41,Z 512.91,A -85,B 0,C 180,E1 25418.783,E2 25418.783} C_VEL
LIN {X 0,Y 635.793,Z 478.953,A -85,B 0,C 180,E1 25418.355,E2 25418.355} C_VEL
LIN {X 0,Y 636.46,Z 469.813,A -85,B 0,C 180,E1 25418.186,E2 25418.186} C_VEL
LIN {X 0,Y 638.707,Z 445.788,A -85,B 0,C 180,E1 25417.794,E2 25417.794} C_VEL
LIN {X 0,Y 639.326,Z 439.697,A -85,B 0,C 180,E1 25417.699,E2 25417.699} C_VEL
LIN {X 0,Y 631.353,Z 430.659,A -85,B 0,C 180,E1 25416.575,E2 25416.575} C_VEL
LIN {X 0,Y 614.277,Z 404.879,A -85,B 0,C 180,E1 25413.771,E2 25413.771} C_VEL
LIN {X 0,Y 603.191,Z 389.133,A -85,B 0,C 180,E1 25411.785,E2 25411.785} C_VEL
LIN {X 0,Y 592.87,Z 374.924,A -85,B 0,C 180,E1 25409.781,E2 25409.781} C_VEL
LIN {X 0,Y 587.925,Z 368.592,A -85,B 0,C 180,E1 25408.771,E2 25408.771} C_VEL
LIN {X 0,Y 584.278,Z 363.827,A -85,B 0,C 180,E1 25407.991,E2 25407.991} C_VEL
LIN {X 0,Y 580.85,Z 359.14,A -85,B 0,C 180,E1 25407.224,E2 25407.224} C_VEL
LIN {X 0,Y 577.017,Z 354.643,A -85,B 0,C 180,E1 25406.362,E2 25406.362} C_VEL
LIN {X 0,Y 575.589,Z 352.586,A -85,B 0,C 180,E1 25406.017,E2 25406.017} C_VEL
LIN {X 0,Y 572.367,Z 348.959,A -85,B 0,C 180,E1 25405.258,E2 25405.258} C_VEL
LIN {X 0,Y 571.034,Z 346.738,A -85,B 0,C 180,E1 25404.905,E2 25404.905} C_VEL
LIN {X 0,Y 567.949,Z 343.82,A -85,B 0,C 180,E1 25404.162,E2 25404.162} C_VEL
LIN {X 0,Y 566.304,Z 340.641,A -85,B 0,C 180,E1 25403.684,E2 25403.684} C_VEL
LIN {X 0,Y 563.161,Z 338.367,A -85,B 0,C 180,E1 25402.91,E2 25402.91} C_VEL
LIN {X 0,Y 561.669,Z 335.509,A -85,B 0,C 180,E1 25402.449,E2 25402.449} C_VEL
LIN {X 0,Y 561.432,Z 334.302,A -85,B 0,C 180,E1 25402.318,E2 25402.318} C_VEL
LIN {X 0,Y 561.413,Z 334.299,A -85,B 0,C 180,E1 25399.13,E2 25399.13} C_VEL
LIN {X 0,Y 561.443,Z 334.29,A -85,B 0,C 180,E1 25395.812,E2 25395.812} C_VEL
LIN {X 0,Y 561.427,Z 334.416,A -85,B 0,C 180,E1 25395.283,E2 25395.283} C_VEL
LIN {X 0,Y 567.923,Z 353.698,A -85,B 0,C 180,E1 25394.336,E2 25394.336} C_VEL
LIN {X 0,Y 567.694,Z 433.256,A -85,B 0,C 180,E1 25391.506,E2 25391.506} C_VEL
LIN {X 0,Y 567.89,Z 512.836,A -85,B 0,C 180,E1 25388.531,E2 25388.531} C_VEL
LIN {X 0,Y 567.727,Z 584.727,A -85,B 0,C 180,E1 25385.762,E2 25385.762} C_VEL
LIN {X 0,Y 567.179,Z 655.072,A -85,B 0,C 180,E1 25382.981,E2 25382.981} C_VEL
LIN {X 0,Y 566.265,Z 736.735,A -85,B 0,C 180,E1 25379.696,E2 25379.696} C_VEL
LIN {X 0,Y 565.179,Z 816.737,A -85,B 0,C 180,E1 25376.399,E2 25376.399} C_VEL
LIN {X 0,Y 564.506,Z 850.105,A -85,B 0,C 180,E1 25375.021,E2 25375.021} C_VEL
LIN {X 0,Y 563.909,Z 858.925,A -85,B 0,C 180,E1 25374.695,E2 25374.695} C_VEL
LIN {X 0,Y 563.169,Z 972.678,A -85,B 0,C 180,E1 25373.139,E2 25373.139} C_VEL
LIN {X 0,Y 563.206,Z 985.227,A -85,B 0,C 180,E1 25372.835,E2 25372.835} C_VEL
LIN {X 0,Y 563.174,Z 996.281,A -85,B 0,C 180,E1 25372.45,E2 25372.45} C_VEL
LIN {X 0,Y 563.052,Z 1008.501,A -85,B 0,C 180,E1 25371.884,E2 25371.884} C_VEL
LIN {X 0,Y 562.809,Z 1022.019,A -85,B 0,C 180,E1 25371.041,E2 25371.041} C_VEL
LIN {X 0,Y 562.566,Z 1032.12,A -85,B 0,C 180,E1 25370.227,E2 25370.227} C_VEL
LIN {X 0,Y 562.334,Z 1040.091,A -85,B 0,C 180,E1 25369.447,E2 25369.447} C_VEL
LIN {X 0,Y 562.079,Z 1048,A -85,B 0,C 180,E1 25368.508,E2 25368.508} C_VEL
LIN {X 0,Y 561.836,Z 1055.15,A -85,B 0,C 180,E1 25367.46,E2 25367.46} C_VEL
LIN {X 0,Y 561.559,Z 1062.598,A -85,B 0,C 180,E1 25366.027,E2 25366.027} C_VEL
LIN {X 0,Y 561.392,Z 1067.099,A -85,B 0,C 180,E1 25364.822,E2 25364.822} C_VEL
LIN {X 0,Y 561.272,Z 1070.184,A -85,B 0,C 180,E1 25363.652,E2 25363.652} C_VEL
LIN {X 0,Y 561.198,Z 1072.09,A -85,B 0,C 180,E1 25362.476,E2 25362.476} C_VEL
LIN {X 0,Y 561.149,Z 1072.886,A -85,B 0,C 180,E1 25361.185,E2 25361.185} C_VEL
LIN {X 0,Y 561.154,Z 1071.937,A -85,B 0,C 180,E1 25359.559,E2 25359.559} C_VEL
LIN {X 0,Y 561.191,Z 1069.563,A -85,B 0,C 180,E1 25358.247,E2 25358.247} C_VEL
LIN {X 0,Y 561.282,Z 1066.095,A -85,B 0,C 180,E1 25357.037,E2 25357.037} C_VEL
LIN {X 0,Y 561.445,Z 1060.756,A -85,B 0,C 180,E1 25355.707,E2 25355.707} C_VEL
LIN {X 0,Y 561.685,Z 1053.368,A -85,B 0,C 180,E1 25354.368,E2 25354.368} C_VEL
LIN {X 0,Y 561.935,Z 1045.697,A -85,B 0,C 180,E1 25353.285,E2 25353.285} C_VEL
LIN {X 0,Y 562.208,Z 1037.016,A -85,B 0,C 180,E1 25352.29,E2 25352.29} C_VEL
LIN {X 0,Y 562.539,Z 1026.18,A -85,B 0,C 180,E1 25351.287,E2 25351.287} C_VEL
LIN {X 0,Y 562.811,Z 1013.768,A -85,B 0,C 180,E1 25350.403,E2 25350.403} C_VEL
LIN {X 0,Y 563.02,Z 1002.861,A -85,B 0,C 180,E1 25349.788,E2 25349.788} C_VEL
LIN {X 0,Y 563.169,Z 991.577,A -85,B 0,C 180,E1 25349.289,E2 25349.289} C_VEL
LIN {X 0,Y 563.269,Z 977.203,A -85,B 0,C 180,E1 25348.823,E2 25348.823} C_VEL
LIN {X 0,Y 563.228,Z 960.268,A -85,B 0,C 180,E1 25348.512,E2 25348.512} C_VEL
LIN {X 0,Y 564.12,Z 852.613,A -85,B 0,C 180,E1 25347.063,E2 25347.063} C_VEL
LIN {X 0,Y 564.779,Z 836.438,A -85,B 0,C 180,E1 25346.381,E2 25346.381} C_VEL
LIN {X 0,Y 566.228,Z 755.868,A -85,B 0,C 180,E1 25342.918,E2 25342.918} C_VEL
LIN {X 0,Y 566.241,Z 755.107,A -85,B 0,C 180,E1 25342.885,E2 25342.885} C_VEL
LIN {X 0,Y 565.378,Z 750.473,A -85,B 0,C 180,E1 25342.654,E2 25342.654} C_VEL
LIN {X 0,Y 559.656,Z 739.047,A -85,B 0,C 180,E1 25341.962,E2 25341.962} C_VEL
LIN {X 0,Y 558.996,Z 735.045,A -85,B 0,C 180,E1 25341.765,E2 25341.765} C_VEL
LIN {X 0,Y 559.18,Z 728.656,A -85,B 0,C 180,E1 25341.468,E2 25341.468} C_VEL
LIN {X 0,Y 560.325,Z 730.096,A -85,B 0,C 180,E1 25341.284,E2 25341.284} C_VEL
LIN {X 0,Y 562.143,Z 729.707,A -85,B 0,C 180,E1 25341.073,E2 25341.073} C_VEL
LIN {X 0,Y 565.057,Z 726.753,A -85,B 0,C 180,E1 25340.807,E2 25340.807} C_VEL
LIN {X 0,Y 568.739,Z 720.817,A -85,B 0,C 180,E1 25340.539,E2 25340.539} C_VEL
LIN {X 0,Y 572.058,Z 719.288,A -85,B 0,C 180,E1 25340.196,E2 25340.196} C_VEL
LIN {X 0,Y 575.981,Z 715.349,A -85,B 0,C 180,E1 25339.857,E2 25339.857} C_VEL
LIN {X 0,Y 579.363,Z 710.606,A -85,B 0,C 180,E1 25339.605,E2 25339.605} C_VEL
LIN {X 0,Y 583.817,Z 707.525,A -85,B 0,C 180,E1 25339.202,E2 25339.202} C_VEL
LIN {X 0,Y 588.407,Z 702.275,A -85,B 0,C 180,E1 25338.848,E2 25338.848} C_VEL
LIN {X 0,Y 590.24,Z 700.027,A -85,B 0,C 180,E1 25338.713,E2 25338.713} C_VEL
LIN {X 0,Y 595.45,Z 695.937,A -85,B 0,C 180,E1 25338.287,E2 25338.287} C_VEL
LIN {X 0,Y 600.67,Z 690.045,A -85,B 0,C 180,E1 25337.926,E2 25337.926} C_VEL
LIN {X 0,Y 595.408,Z 815.107,A -85,B 0,C 180,E1 25335.918,E2 25335.918} C_VEL
LIN {X 0,Y 593.758,Z 841.911,A -85,B 0,C 180,E1 25335.323,E2 25335.323} C_VEL
LIN {X 0,Y 592.068,Z 864.574,A -85,B 0,C 180,E1 25334.694,E2 25334.694} C_VEL
LIN {X 0,Y 589.525,Z 893.631,A -85,B 0,C 180,E1 25333.692,E2 25333.692} C_VEL
LIN {X 0,Y 587.061,Z 918.011,A -85,B 0,C 180,E1 25332.679,E2 25332.679} C_VEL
LIN {X 0,Y 584.122,Z 943.406,A -85,B 0,C 180,E1 25331.43,E2 25331.43} C_VEL
LIN {X 0,Y 581.002,Z 966.784,A -85,B 0,C 180,E1 25330.065,E2 25330.065} C_VEL
LIN {X 0,Y 578.098,Z 987.05,A -85,B 0,C 180,E1 25328.708,E2 25328.708} C_VEL
LIN {X 0,Y 575.89,Z 1001.642,A -85,B 0,C 180,E1 25327.611,E2 25327.611} C_VEL
LIN {X 0,Y 572.754,Z 1019.224,A -85,B 0,C 180,E1 25326.071,E2 25326.071} C_VEL
LIN {X 0,Y 569.707,Z 1036.18,A -85,B 0,C 180,E1 25324.413,E2 25324.413} C_VEL
LIN {X 0,Y 566.84,Z 1052.235,A -85,B 0,C 180,E1 25322.669,E2 25322.669} C_VEL
LIN {X 0,Y 564.141,Z 1067.636,A -85,B 0,C 180,E1 25320.813,E2 25320.813} C_VEL
LIN {X 0,Y 561.337,Z 1084.689,A -85,B 0,C 180,E1 25318.515,E2 25318.515} C_VEL
LIN {X 0,Y 558.73,Z 1100.931,A -85,B 0,C 180,E1 25316.006,E2 25316.006} C_VEL
LIN {X 0,Y 556.935,Z 1113.415,A -85,B 0,C 180,E1 25313.826,E2 25313.826} C_VEL
LIN {X 0,Y 555.558,Z 1123.987,A -85,B 0,C 180,E1 25311.763,E2 25311.763} C_VEL
LIN {X 0,Y 554.466,Z 1133.392,A -85,B 0,C 180,E1 25309.709,E2 25309.709} C_VEL
LIN {X 0,Y 553.576,Z 1142.114,A -85,B 0,C 180,E1 25307.557,E2 25307.557} C_VEL
LIN {X 0,Y 552.942,Z 1149.702,A -85,B 0,C 180,E1 25305.417,E2 25305.417} C_VEL
LIN {X 0,Y 552.489,Z 1156.546,A -85,B 0,C 180,E1 25303.176,E2 25303.176} C_VEL
LIN {X 0,Y 552.167,Z 1162.705,A -85,B 0,C 180,E1 25300.751,E2 25300.751} C_VEL
LIN {X 0,Y 552.011,Z 1167.789,A -85,B 0,C 180,E1 25298.228,E2 25298.228} C_VEL
LIN {X 0,Y 551.928,Z 1171.991,A -85,B 0,C 180,E1 25295.302,E2 25295.302} C_VEL
LIN {X 0,Y 551.908,Z 1174.152,A -85,B 0,C 180,E1 25292.701,E2 25292.701} C_VEL
LIN {X 0,Y 551.897,Z 1174.915,A -85,B 0,C 180,E1 25290.313,E2 25290.313} C_VEL
LIN {X 0,Y 551.911,Z 1174.439,A -85,B 0,C 180,E1 25287.821,E2 25287.821} C_VEL
LIN {X 0,Y 551.918,Z 1172.867,A -85,B 0,C 180,E1 25285.533,E2 25285.533} C_VEL
LIN {X 0,Y 551.951,Z 1170.189,A -85,B 0,C 180,E1 25283.239,E2 25283.239} C_VEL
LIN {X 0,Y 552.041,Z 1166.388,A -85,B 0,C 180,E1 25280.935,E2 25280.935} C_VEL
LIN {X 0,Y 552.202,Z 1161.683,A -85,B 0,C 180,E1 25278.724,E2 25278.724} C_VEL
LIN {X 0,Y 552.548,Z 1155.464,A -85,B 0,C 180,E1 25276.351,E2 25276.351} C_VEL
LIN {X 0,Y 553.075,Z 1147.887,A -85,B 0,C 180,E1 25273.944,E2 25273.944} C_VEL
LIN {X 0,Y 554.106,Z 1136.863,A -85,B 0,C 180,E1 25271.009,E2 25271.009} C_VEL
LIN {X 0,Y 555.315,Z 1125.986,A -85,B 0,C 180,E1 25268.562,E2 25268.562} C_VEL
LIN {X 0,Y 556.628,Z 1115.647,A -85,B 0,C 180,E1 25266.499,E2 25266.499} C_VEL
LIN {X 0,Y 558.273,Z 1104.054,A -85,B 0,C 180,E1 25264.43,E2 25264.43} C_VEL
LIN {X 0,Y 560.128,Z 1091.81,A -85,B 0,C 180,E1 25262.463,E2 25262.463} C_VEL
LIN {X 0,Y 562.339,Z 1078.206,A -85,B 0,C 180,E1 25260.495,E2 25260.495} C_VEL
LIN {X 0,Y 564.954,Z 1063.087,A -85,B 0,C 180,E1 25258.528,E2 25258.528} C_VEL
LIN {X 0,Y 568.49,Z 1043.307,A -85,B 0,C 180,E1 25256.236,E2 25256.236} C_VEL
LIN {X 0,Y 571.916,Z 1023.871,A -85,B 0,C 180,E1 25254.274,E2 25254.274} C_VEL
LIN {X 0,Y 575.022,Z 1006.452,A -85,B 0,C 180,E1 25252.702,E2 25252.702} C_VEL
LIN {X 0,Y 577.285,Z 992.813,A -85,B 0,C 180,E1 25251.617,E2 25251.617} C_VEL
LIN {X 0,Y 580.478,Z 970.595,A -85,B 0,C 180,E1 25250.088,E2 25250.088} C_VEL
LIN {X 0,Y 583.358,Z 949.201,A -85,B 0,C 180,E1 25248.804,E2 25248.804} C_VEL
LIN {X 0,Y 585.461,Z 932.281,A -85,B 0,C 180,E1 25247.909,E2 25247.909} C_VEL
LIN {X 0,Y 587.596,Z 912.813,A -85,B 0,C 180,E1 25247.009,E2 25247.009} C_VEL
LIN {X 0,Y 589.837,Z 890.31,A -85,B 0,C 180,E1 25246.093,E2 25246.093} C_VEL
LIN {X 0,Y 592.164,Z 863.139,A -85,B 0,C 180,E1 25245.176,E2 25245.176} C_VEL
LIN {X 0,Y 593.729,Z 842.205,A -85,B 0,C 180,E1 25244.596,E2 25244.596} C_VEL
LIN {X 0,Y 595.096,Z 819.779,A -85,B 0,C 180,E1 25244.093,E2 25244.093} C_VEL
LIN {X 0,Y 596.456,Z 792.412,A -85,B 0,C 180,E1 25243.611,E2 25243.611} C_VEL
LIN {X 0,Y 600.364,Z 696.107,A -85,B 0,C 180,E1 25242.086,E2 25242.086} C_VEL
LIN {X 0,Y 609.653,Z 518.1,A -85,B 0,C 180,E1 25239.166,E2 25239.166} C_VEL
LIN {X 0,Y 614.048,Z 417.115,A -85,B 0,C 180,E1 25237.62,E2 25237.62} C_VEL
LIN {X 0,Y 613.984,Z 415.52,A -85,B 0,C 180,E1 25237.581,E2 25237.581} C_VEL
LIN {X 0,Y 600.49,Z 402.505,A -85,B 0,C 180,E1 25235.589,E2 25235.589} C_VEL
LIN {X 0,Y 592.537,Z 395.362,A -85,B 0,C 180,E1 25234.336,E2 25234.336} C_VEL
LIN {X 0,Y 585.441,Z 388.938,A -85,B 0,C 180,E1 25233.13,E2 25233.13} C_VEL
LIN {X 0,Y 583.079,Z 384.456,A -85,B 0,C 180,E1 25231.536,E2 25231.536} C_VEL
LIN {X 0,Y 580.814,Z 380.043,A -85,B 0,C 180,E1 25229.817,E2 25229.817} C_VEL
LIN {X 0,Y 578.178,Z 375.642,A -85,B 0,C 180,E1 25227.724,E2 25227.724} C_VEL
LIN {X 0,Y 577.483,Z 374.394,A -85,B 0,C 180,E1 25227.089,E2 25227.089} C_VEL
LIN {X 0,Y 575.197,Z 370.398,A -85,B 0,C 180,E1 25224.768,E2 25224.768} C_VEL
LIN {X 0,Y 574.718,Z 369.336,A -85,B 0,C 180,E1 25224.133,E2 25224.133} C_VEL
LIN {X 0,Y 572.047,Z 364.714,A -85,B 0,C 180,E1 25220.142,E2 25220.142} C_VEL
LIN {X 0,Y 571.49,Z 363.869,A -85,B 0,C 180,E1 25218.992,E2 25218.992} C_VEL
LIN {X 0,Y 570.247,Z 362.631,A -85,B 0,C 180,E1 25214.566,E2 25214.566} C_VEL
LIN {X 0,Y 570.897,Z 363.338,A -85,B 0,C 180,E1 25210.597,E2 25210.597} C_VEL
LIN {X 0,Y 572.063,Z 364.6,A -85,B 0,C 180,E1 25208.24,E2 25208.24} C_VEL
LIN {X 0,Y 575.233,Z 370.054,A -85,B 0,C 180,E1 25203.688,E2 25203.688} C_VEL
LIN {X 0,Y 577.379,Z 374.206,A -85,B 0,C 180,E1 25201.389,E2 25201.389} C_VEL
LIN {X 0,Y 578.261,Z 375.397,A -85,B 0,C 180,E1 25200.694,E2 25200.694} C_VEL
LIN {X 0,Y 580.509,Z 379.539,A -85,B 0,C 180,E1 25198.816,E2 25198.816} C_VEL
LIN {X 0,Y 581.41,Z 381.198,A -85,B 0,C 180,E1 25198.127,E2 25198.127} C_VEL
LIN {X 0,Y 584.099,Z 385.983,A -85,B 0,C 180,E1 25196.27,E2 25196.27} C_VEL
LIN {X 0,Y 586.865,Z 391.064,A -85,B 0,C 180,E1 25194.525,E2 25194.525} C_VEL
LIN {X 0,Y 589.659,Z 396.361,A -85,B 0,C 180,E1 25192.889,E2 25192.889} C_VEL
LIN {X 0,Y 592.32,Z 401.357,A -85,B 0,C 180,E1 25191.457,E2 25191.457} C_VEL
LIN {X 0,Y 596.495,Z 409.315,A -85,B 0,C 180,E1 25189.374,E2 25189.374} C_VEL
LIN {X 0,Y 602.586,Z 421.558,A -85,B 0,C 180,E1 25186.567,E2 25186.567} C_VEL
LIN {X 0,Y 608.628,Z 434.507,A -85,B 0,C 180,E1 25183.978,E2 25183.978} C_VEL
LIN {X 0,Y 610.313,Z 438.212,A -85,B 0,C 180,E1 25183.29,E2 25183.29} C_VEL
LIN {X 0,Y 605.418,Z 471.202,A -85,B 0,C 180,E1 25180.461,E2 25180.461} C_VEL
LIN {X 0,Y 600.624,Z 505.55,A -85,B 0,C 180,E1 25177.642,E2 25177.642} C_VEL
LIN {X 0,Y 595.88,Z 542.146,A -85,B 0,C 180,E1 25174.744,E2 25174.744} C_VEL
LIN {X 0,Y 590.422,Z 591.828,A -85,B 0,C 180,E1 25170.906,E2 25170.906} C_VEL
